      movel([0.367168, -1.380933, -2.569217, -0.762240, 1.570796, 1.937965],accel_mss,speed_ms,0,blend_radius_m)
      movel([0.367388, -1.380879, -2.569255, -0.762256, 1.570796, 1.938184],accel_mss,speed_ms,0,blend_radius_m)
      movel([0.367623, -1.380831, -2.569289, -0.762270, 1.570796, 1.938419],accel_mss,speed_ms,0,blend_radius_m)
      movel([0.367853, -1.380796, -2.569313, -0.762280, 1.570796, 1.938649],accel_mss,speed_ms,0,blend_radius_m)
      movel([0.368080, -1.380773, -2.569329, -0.762287, 1.570796, 1.938877],accel_mss,speed_ms,0,blend_radius_m)
      movel([0.368708, -1.380733, -2.569357, -0.762298, 1.570796, 1.939505],accel_mss,speed_ms,0,blend_radius_m)
      movel([0.369332, -1.380703, -2.569379, -0.762307, 1.570796, 1.940129],accel_mss,speed_ms,0,blend_radius_m)
      movel([0.369955, -1.380682, -2.569394, -0.762313, 1.570796, 1.940751],accel_mss,speed_ms,0,blend_radius_m)
      movel([0.370572, -1.380670, -2.569402, -0.762317, 1.570796, 1.941368],accel_mss,speed_ms,0,blend_radius_m)
      movel([0.370788, -1.380675, -2.569399, -0.762315, 1.570796, 1.941585],accel_mss,speed_ms,0,blend_radius_m)
      movel([0.370998, -1.380691, -2.569387, -0.762311, 1.570796, 1.941795],accel_mss,speed_ms,0,blend_radius_m)
      movel([0.371200, -1.380721, -2.569366, -0.762302, 1.570796, 1.941996],accel_mss,speed_ms,0,blend_radius_m)
      movel([0.371383, -1.380759, -2.569339, -0.762291, 1.570796, 1.942179],accel_mss,speed_ms,0,blend_radius_m)
      movel([0.371557, -1.380812, -2.569302, -0.762275, 1.570796, 1.942353],accel_mss,speed_ms,0,blend_radius_m)
      movel([0.371719, -1.380877, -2.569256, -0.762256, 1.570796, 1.942516],accel_mss,speed_ms,0,blend_radius_m)
      movel([0.372096, -1.381057, -2.569129, -0.762203, 1.570796, 1.942892],accel_mss,speed_ms,0,blend_radius_m)
      movel([0.372463, -1.381249, -2.568993, -0.762147, 1.570796, 1.943259],accel_mss,speed_ms,0,blend_radius_m)
      movel([0.372728, -1.381406, -2.568882, -0.762101, 1.570796, 1.943524],accel_mss,speed_ms,0,blend_radius_m)
      movel([0.372979, -1.381575, -2.568762, -0.762052, 1.570796, 1.943776],accel_mss,speed_ms,0,blend_radius_m)
      movel([0.373219, -1.381756, -2.568634, -0.761999, 1.570796, 1.944015],accel_mss,speed_ms,0,blend_radius_m)
      movel([0.373443, -1.381953, -2.568494, -0.761941, 1.570796, 1.944239],accel_mss,speed_ms,0,blend_radius_m)
      movel([0.373656, -1.382160, -2.568348, -0.761881, 1.570796, 1.944452],accel_mss,speed_ms,0,blend_radius_m)
      movel([0.373848, -1.382378, -2.568193, -0.761818, 1.570796, 1.944644],accel_mss,speed_ms,0,blend_radius_m)
      movel([0.374028, -1.382608, -2.568030, -0.761751, 1.570796, 1.944825],accel_mss,speed_ms,0,blend_radius_m)
      movel([0.374190, -1.382850, -2.567859, -0.761681, 1.570796, 1.944986],accel_mss,speed_ms,0,blend_radius_m)
      movel([0.374338, -1.383103, -2.567679, -0.761607, 1.570796, 1.945134],accel_mss,speed_ms,0,blend_radius_m)
      movel([0.374468, -1.383366, -2.567492, -0.761531, 1.570796, 1.945264],accel_mss,speed_ms,0,blend_radius_m)
      movel([0.374585, -1.383643, -2.567295, -0.761451, 1.570796, 1.945381],accel_mss,speed_ms,0,blend_radius_m)
      movel([0.374684, -1.383931, -2.567090, -0.761368, 1.570796, 1.945480],accel_mss,speed_ms,0,blend_radius_m)
      movel([0.374766, -1.384226, -2.566880, -0.761282, 1.570796, 1.945562],accel_mss,speed_ms,0,blend_radius_m)
      movel([0.374834, -1.384529, -2.566665, -0.761195, 1.570796, 1.945630],accel_mss,speed_ms,0,blend_radius_m)
      movel([0.374881, -1.384841, -2.566442, -0.761105, 1.570796, 1.945678],accel_mss,speed_ms,0,blend_radius_m)
      movel([0.374915, -1.385171, -2.566207, -0.761011, 1.570796, 1.945711],accel_mss,speed_ms,0,blend_radius_m)
      movel([0.374934, -1.385509, -2.565967, -0.760914, 1.570796, 1.945730],accel_mss,speed_ms,0,blend_radius_m)
      movel([0.374935, -1.385851, -2.565722, -0.760816, 1.570796, 1.945731],accel_mss,speed_ms,0,blend_radius_m)
      movel([0.374922, -1.386197, -2.565475, -0.760717, 1.570796, 1.945718],accel_mss,speed_ms,0,blend_radius_m)
      movel([0.374892, -1.386549, -2.565223, -0.760617, 1.570796, 1.945688],accel_mss,speed_ms,0,blend_radius_m)
      movel([0.374857, -1.386821, -2.565029, -0.760539, 1.570796, 1.945653],accel_mss,speed_ms,0,blend_radius_m)
      movel([0.374809, -1.387098, -2.564831, -0.760461, 1.570796, 1.945605],accel_mss,speed_ms,0,blend_radius_m)
      movel([0.374747, -1.387375, -2.564633, -0.760382, 1.570796, 1.945543],accel_mss,speed_ms,0,blend_radius_m)
      movel([0.374671, -1.387656, -2.564431, -0.760302, 1.570796, 1.945468],accel_mss,speed_ms,0,blend_radius_m)
      movel([0.374535, -1.388106, -2.564108, -0.760175, 1.570796, 1.945331],accel_mss,speed_ms,0,blend_radius_m)
      movel([0.374382, -1.388556, -2.563786, -0.760048, 1.570796, 1.945178],accel_mss,speed_ms,0,blend_radius_m)
      movel([0.374215, -1.389008, -2.563461, -0.759920, 1.570796, 1.945011],accel_mss,speed_ms,0,blend_radius_m)
      movel([0.374032, -1.389458, -2.563137, -0.759794, 1.570796, 1.944829],accel_mss,speed_ms,0,blend_radius_m)
      movel([0.373834, -1.389909, -2.562813, -0.759667, 1.570796, 1.944630],accel_mss,speed_ms,0,blend_radius_m)
      movel([0.373623, -1.390357, -2.562490, -0.759542, 1.570796, 1.944419],accel_mss,speed_ms,0,blend_radius_m)
      movel([0.373481, -1.390635, -2.562289, -0.759464, 1.570796, 1.944277],accel_mss,speed_ms,0,blend_radius_m)
      movel([0.373327, -1.390909, -2.562092, -0.759388, 1.570796, 1.944123],accel_mss,speed_ms,0,blend_radius_m)
      movel([0.373162, -1.391181, -2.561896, -0.759312, 1.570796, 1.943958],accel_mss,speed_ms,0,blend_radius_m)
      movel([0.372986, -1.391454, -2.561699, -0.759236, 1.570796, 1.943782],accel_mss,speed_ms,0,blend_radius_m)
      movel([0.372747, -1.391796, -2.561451, -0.759141, 1.570796, 1.943544],accel_mss,speed_ms,0,blend_radius_m)
      movel([0.372498, -1.392137, -2.561205, -0.759047, 1.570796, 1.943295],accel_mss,speed_ms,0,blend_radius_m)
      movel([0.372235, -1.392473, -2.560962, -0.758954, 1.570796, 1.943032],accel_mss,speed_ms,0,blend_radius_m)
      movel([0.371963, -1.392805, -2.560722, -0.758862, 1.570796, 1.942759],accel_mss,speed_ms,0,blend_radius_m)
      movel([0.371681, -1.393131, -2.560486, -0.758772, 1.570796, 1.942478],accel_mss,speed_ms,0,blend_radius_m)
      movel([0.371388, -1.393453, -2.560253, -0.758684, 1.570796, 1.942184],accel_mss,speed_ms,0,blend_radius_m)
      movel([0.371084, -1.393768, -2.560024, -0.758597, 1.570796, 1.941880],accel_mss,speed_ms,0,blend_radius_m)
      movel([0.370782, -1.394067, -2.559806, -0.758515, 1.570796, 1.941578],accel_mss,speed_ms,0,blend_radius_m)
      movel([0.370466, -1.394361, -2.559593, -0.758435, 1.570796, 1.941263],accel_mss,speed_ms,0,blend_radius_m)
      movel([0.370145, -1.394648, -2.559385, -0.758356, 1.570796, 1.940941],accel_mss,speed_ms,0,blend_radius_m)
      movel([0.369814, -1.394924, -2.559184, -0.758281, 1.570796, 1.940610],accel_mss,speed_ms,0,blend_radius_m)
      movel([0.369476, -1.395194, -2.558987, -0.758207, 1.570796, 1.940273],accel_mss,speed_ms,0,blend_radius_m)
      movel([0.369130, -1.395453, -2.558799, -0.758137, 1.570796, 1.939926],accel_mss,speed_ms,0,blend_radius_m)
      movel([0.368780, -1.395704, -2.558616, -0.758069, 1.570796, 1.939577],accel_mss,speed_ms,0,blend_radius_m)
      movel([0.368427, -1.395942, -2.558443, -0.758004, 1.570796, 1.939223],accel_mss,speed_ms,0,blend_radius_m)
      movel([0.368069, -1.396168, -2.558278, -0.757943, 1.570796, 1.938865],accel_mss,speed_ms,0,blend_radius_m)
      movel([0.367709, -1.396384, -2.558121, -0.757884, 1.570796, 1.938505],accel_mss,speed_ms,0,blend_radius_m)
      movel([0.367343, -1.396587, -2.557972, -0.757829, 1.570796, 1.938139],accel_mss,speed_ms,0,blend_radius_m)
      movel([0.366973, -1.396782, -2.557831, -0.757777, 1.570796, 1.937769],accel_mss,speed_ms,0,blend_radius_m)
      movel([0.366600, -1.396963, -2.557698, -0.757728, 1.570796, 1.937396],accel_mss,speed_ms,0,blend_radius_m)
      movel([0.366227, -1.397132, -2.557575, -0.757682, 1.570796, 1.937023],accel_mss,speed_ms,0,blend_radius_m)
      movel([0.365850, -1.397290, -2.557460, -0.757640, 1.570796, 1.936646],accel_mss,speed_ms,0,blend_radius_m)
      movel([0.365473, -1.397434, -2.557354, -0.757601, 1.570796, 1.936270],accel_mss,speed_ms,0,blend_radius_m)
      movel([0.365097, -1.397568, -2.557256, -0.757565, 1.570796, 1.935893],accel_mss,speed_ms,0,blend_radius_m)
      movel([0.364719, -1.397687, -2.557169, -0.757533, 1.570796, 1.935516],accel_mss,speed_ms,0,blend_radius_m)
      movel([0.364343, -1.397793, -2.557092, -0.757504, 1.570796, 1.935139],accel_mss,speed_ms,0,blend_radius_m)
      movel([0.363969, -1.397886, -2.557024, -0.757479, 1.570796, 1.934766],accel_mss,speed_ms,0,blend_radius_m)
      movel([0.363599, -1.397965, -2.556966, -0.757458, 1.570796, 1.934395],accel_mss,speed_ms,0,blend_radius_m)
      movel([0.363252, -1.398025, -2.556922, -0.757442, 1.570796, 1.934048],accel_mss,speed_ms,0,blend_radius_m)
      movel([0.362911, -1.398069, -2.556890, -0.757430, 1.570796, 1.933708],accel_mss,speed_ms,0,blend_radius_m)
      movel([0.362576, -1.398099, -2.556868, -0.757422, 1.570796, 1.933372],accel_mss,speed_ms,0,blend_radius_m)
      movel([0.362245, -1.398113, -2.556858, -0.757418, 1.570796, 1.933042],accel_mss,speed_ms,0,blend_radius_m)
      movel([0.361921, -1.398111, -2.556859, -0.757419, 1.570796, 1.932717],accel_mss,speed_ms,0,blend_radius_m)
      movel([0.361603, -1.398095, -2.556871, -0.757423, 1.570796, 1.932400],accel_mss,speed_ms,0,blend_radius_m)
      movel([0.361295, -1.398062, -2.556895, -0.757432, 1.570796, 1.932092],accel_mss,speed_ms,0,blend_radius_m)
      movel([0.360993, -1.398014, -2.556930, -0.757445, 1.570796, 1.931790],accel_mss,speed_ms,0,blend_radius_m)
      movel([0.360704, -1.397950, -2.556977, -0.757462, 1.570796, 1.931501],accel_mss,speed_ms,0,blend_radius_m)
      movel([0.360408, -1.397869, -2.557036, -0.757484, 1.570796, 1.931204],accel_mss,speed_ms,0,blend_radius_m)
      movel([0.360124, -1.397775, -2.557105, -0.757509, 1.570796, 1.930920],accel_mss,speed_ms,0,blend_radius_m)
      movel([0.359848, -1.397665, -2.557185, -0.757539, 1.570796, 1.930645],accel_mss,speed_ms,0,blend_radius_m)
      movel([0.359584, -1.397544, -2.557274, -0.757571, 1.570796, 1.930380],accel_mss,speed_ms,0,blend_radius_m)
      movel([0.359331, -1.397409, -2.557372, -0.757607, 1.570796, 1.930127],accel_mss,speed_ms,0,blend_radius_m)
      movel([0.359090, -1.397261, -2.557481, -0.757647, 1.570796, 1.929886],accel_mss,speed_ms,0,blend_radius_m)
      movel([0.358861, -1.397102, -2.557597, -0.757690, 1.570796, 1.929657],accel_mss,speed_ms,0,blend_radius_m)
      movel([0.358643, -1.396929, -2.557723, -0.757737, 1.570796, 1.929439],accel_mss,speed_ms,0,blend_radius_m)
      movel([0.358439, -1.396744, -2.557858, -0.757787, 1.570796, 1.929235],accel_mss,speed_ms,0,blend_radius_m)
      movel([0.358240, -1.396540, -2.558007, -0.757842, 1.570796, 1.929036],accel_mss,speed_ms,0,blend_radius_m)
      movel([0.358054, -1.396325, -2.558164, -0.757900, 1.570796, 1.928851],accel_mss,speed_ms,0,blend_radius_m)
      movel([0.357880, -1.396097, -2.558330, -0.757962, 1.570796, 1.928676],accel_mss,speed_ms,0,blend_radius_m)
      movel([0.357724, -1.395859, -2.558504, -0.758027, 1.570796, 1.928520],accel_mss,speed_ms,0,blend_radius_m)
      movel([0.357580, -1.395611, -2.558684, -0.758094, 1.570796, 1.928376],accel_mss,speed_ms,0,blend_radius_m)
      movel([0.357451, -1.395353, -2.558872, -0.758164, 1.570796, 1.928248],accel_mss,speed_ms,0,blend_radius_m)
      movel([0.357335, -1.395086, -2.559066, -0.758237, 1.570796, 1.928131],accel_mss,speed_ms,0,blend_radius_m)
      movel([0.357235, -1.394812, -2.559265, -0.758311, 1.570796, 1.928032],accel_mss,speed_ms,0,blend_radius_m)
      movel([0.357151, -1.394526, -2.559473, -0.758390, 1.570796, 1.927948],accel_mss,speed_ms,0,blend_radius_m)
      movel([0.357072, -1.394192, -2.559716, -0.758481, 1.570796, 1.927869],accel_mss,speed_ms,0,blend_radius_m)
      movel([0.357015, -1.393848, -2.559966, -0.758575, 1.570796, 1.927812],accel_mss,speed_ms,0,blend_radius_m)
      movel([0.356975, -1.393496, -2.560221, -0.758672, 1.570796, 1.927771],accel_mss,speed_ms,0,blend_radius_m)
      movel([0.356953, -1.393135, -2.560483, -0.758771, 1.570796, 1.927750],accel_mss,speed_ms,0,blend_radius_m)
      movel([0.356951, -1.392766, -2.560750, -0.758873, 1.570796, 1.927748],accel_mss,speed_ms,0,blend_radius_m)
      movel([0.356969, -1.392391, -2.561021, -0.758976, 1.570796, 1.927766],accel_mss,speed_ms,0,blend_radius_m)
      movel([0.357005, -1.392011, -2.561296, -0.759082, 1.570796, 1.927802],accel_mss,speed_ms,0,blend_radius_m)
      movel([0.357062, -1.391624, -2.561576, -0.759189, 1.570796, 1.927859],accel_mss,speed_ms,0,blend_radius_m)
      movel([0.357124, -1.391284, -2.561822, -0.759284, 1.570796, 1.927920],accel_mss,speed_ms,0,blend_radius_m)
      movel([0.357196, -1.390939, -2.562071, -0.759380, 1.570796, 1.927992],accel_mss,speed_ms,0,blend_radius_m)
      movel([0.357278, -1.390593, -2.562320, -0.759476, 1.570796, 1.928074],accel_mss,speed_ms,0,blend_radius_m)
      speed_ms = 0.003
      movel([0.357278, -1.393848, -2.563790, -0.754751, 1.570796, 1.928074],accel_mss,speed_ms,0,blend_radius_m)
      speed_ms = 0.007
      movel([0.357356, -1.393564, -2.563996, -0.754829, 1.570796, 1.928153],accel_mss,speed_ms,0,blend_radius_m)
      movel([0.357448, -1.393275, -2.564205, -0.754909, 1.570796, 1.928245],accel_mss,speed_ms,0,blend_radius_m)
      movel([0.357553, -1.392988, -2.564413, -0.754988, 1.570796, 1.928350],accel_mss,speed_ms,0,blend_radius_m)
      movel([0.357672, -1.392700, -2.564621, -0.755068, 1.570796, 1.928469],accel_mss,speed_ms,0,blend_radius_m)
      movel([0.357806, -1.392409, -2.564831, -0.755149, 1.570796, 1.928603],accel_mss,speed_ms,0,blend_radius_m)
      movel([0.357953, -1.392121, -2.565039, -0.755229, 1.570796, 1.928749],accel_mss,speed_ms,0,blend_radius_m)
      movel([0.358142, -1.391770, -2.565292, -0.755327, 1.570796, 1.928938],accel_mss,speed_ms,0,blend_radius_m)
      movel([0.358341, -1.391418, -2.565546, -0.755425, 1.570796, 1.929137],accel_mss,speed_ms,0,blend_radius_m)
      movel([0.358546, -1.391068, -2.565798, -0.755522, 1.570796, 1.929342],accel_mss,speed_ms,0,blend_radius_m)
      movel([0.358793, -1.390674, -2.566082, -0.755633, 1.570796, 1.929589],accel_mss,speed_ms,0,blend_radius_m)
      movel([0.359056, -1.390281, -2.566365, -0.755743, 1.570796, 1.929853],accel_mss,speed_ms,0,blend_radius_m)
      movel([0.359336, -1.389894, -2.566643, -0.755852, 1.570796, 1.930132],accel_mss,speed_ms,0,blend_radius_m)
      movel([0.359627, -1.389510, -2.566919, -0.755960, 1.570796, 1.930424],accel_mss,speed_ms,0,blend_radius_m)
      movel([0.359936, -1.389130, -2.567192, -0.756067, 1.570796, 1.930733],accel_mss,speed_ms,0,blend_radius_m)
      movel([0.360247, -1.388769, -2.567451, -0.756169, 1.570796, 1.931043],accel_mss,speed_ms,0,blend_radius_m)
      movel([0.360574, -1.388414, -2.567705, -0.756269, 1.570796, 1.931370],accel_mss,speed_ms,0,blend_radius_m)
      movel([0.360915, -1.388065, -2.567955, -0.756368, 1.570796, 1.931711],accel_mss,speed_ms,0,blend_radius_m)
      movel([0.361265, -1.387726, -2.568198, -0.756465, 1.570796, 1.932062],accel_mss,speed_ms,0,blend_radius_m)
      movel([0.361629, -1.387396, -2.568435, -0.756559, 1.570796, 1.932425],accel_mss,speed_ms,0,blend_radius_m)
      movel([0.361998, -1.387082, -2.568659, -0.756648, 1.570796, 1.932794],accel_mss,speed_ms,0,blend_radius_m)
      movel([0.362374, -1.386777, -2.568876, -0.756735, 1.570796, 1.933171],accel_mss,speed_ms,0,blend_radius_m)
      movel([0.362763, -1.386485, -2.569085, -0.756819, 1.570796, 1.933559],accel_mss,speed_ms,0,blend_radius_m)
      movel([0.363157, -1.386205, -2.569285, -0.756899, 1.570796, 1.933954],accel_mss,speed_ms,0,blend_radius_m)
      movel([0.363562, -1.385937, -2.569476, -0.756976, 1.570796, 1.934358],accel_mss,speed_ms,0,blend_radius_m)
      movel([0.363972, -1.385683, -2.569657, -0.757049, 1.570796, 1.934768],accel_mss,speed_ms,0,blend_radius_m)
      movel([0.364386, -1.385443, -2.569828, -0.757118, 1.570796, 1.935183],accel_mss,speed_ms,0,blend_radius_m)
      movel([0.364807, -1.385215, -2.569990, -0.757183, 1.570796, 1.935604],accel_mss,speed_ms,0,blend_radius_m)
      movel([0.365231, -1.385005, -2.570140, -0.757244, 1.570796, 1.936027],accel_mss,speed_ms,0,blend_radius_m)
      movel([0.365658, -1.384809, -2.570280, -0.757301, 1.570796, 1.936454],accel_mss,speed_ms,0,blend_radius_m)
      movel([0.366192, -1.384581, -2.570442, -0.757366, 1.570796, 1.936988],accel_mss,speed_ms,0,blend_radius_m)
      movel([0.366727, -1.384364, -2.570596, -0.757429, 1.570796, 1.937523],accel_mss,speed_ms,0,blend_radius_m)
      movel([0.366947, -1.384283, -2.570653, -0.757452, 1.570796, 1.937744],accel_mss,speed_ms,0,blend_radius_m)
      movel([0.367168, -1.384214, -2.570703, -0.757473, 1.570796, 1.937965],accel_mss,speed_ms,0,blend_radius_m)
      movel([0.367388, -1.384160, -2.570741, -0.757488, 1.570796, 1.938184],accel_mss,speed_ms,0,blend_radius_m)
      movel([0.367623, -1.384112, -2.570775, -0.757502, 1.570796, 1.938419],accel_mss,speed_ms,0,blend_radius_m)
      movel([0.367853, -1.384078, -2.570799, -0.757512, 1.570796, 1.938649],accel_mss,speed_ms,0,blend_radius_m)
      movel([0.368080, -1.384055, -2.570816, -0.757519, 1.570796, 1.938877],accel_mss,speed_ms,0,blend_radius_m)
      movel([0.368708, -1.384015, -2.570844, -0.757530, 1.570796, 1.939505],accel_mss,speed_ms,0,blend_radius_m)
      movel([0.369332, -1.383985, -2.570865, -0.757539, 1.570796, 1.940129],accel_mss,speed_ms,0,blend_radius_m)
      movel([0.369955, -1.383964, -2.570880, -0.757545, 1.570796, 1.940751],accel_mss,speed_ms,0,blend_radius_m)
      movel([0.370572, -1.383952, -2.570888, -0.757548, 1.570796, 1.941368],accel_mss,speed_ms,0,blend_radius_m)
      movel([0.370788, -1.383957, -2.570885, -0.757547, 1.570796, 1.941585],accel_mss,speed_ms,0,blend_radius_m)
      movel([0.370998, -1.383973, -2.570874, -0.757542, 1.570796, 1.941795],accel_mss,speed_ms,0,blend_radius_m)
      movel([0.371200, -1.384003, -2.570852, -0.757534, 1.570796, 1.941996],accel_mss,speed_ms,0,blend_radius_m)
      movel([0.371383, -1.384040, -2.570826, -0.757523, 1.570796, 1.942179],accel_mss,speed_ms,0,blend_radius_m)
      movel([0.371557, -1.384094, -2.570788, -0.757507, 1.570796, 1.942353],accel_mss,speed_ms,0,blend_radius_m)
      movel([0.371719, -1.384159, -2.570742, -0.757489, 1.570796, 1.942516],accel_mss,speed_ms,0,blend_radius_m)
      movel([0.372096, -1.384338, -2.570614, -0.757437, 1.570796, 1.942892],accel_mss,speed_ms,0,blend_radius_m)
      movel([0.372463, -1.384529, -2.570479, -0.757381, 1.570796, 1.943259],accel_mss,speed_ms,0,blend_radius_m)
      movel([0.372728, -1.384686, -2.570367, -0.757336, 1.570796, 1.943524],accel_mss,speed_ms,0,blend_radius_m)
      movel([0.372979, -1.384855, -2.570247, -0.757287, 1.570796, 1.943776],accel_mss,speed_ms,0,blend_radius_m)
      movel([0.373219, -1.385035, -2.570119, -0.757235, 1.570796, 1.944015],accel_mss,speed_ms,0,blend_radius_m)
      movel([0.373443, -1.385231, -2.569979, -0.757179, 1.570796, 1.944239],accel_mss,speed_ms,0,blend_radius_m)
      movel([0.373656, -1.385437, -2.569832, -0.757119, 1.570796, 1.944452],accel_mss,speed_ms,0,blend_radius_m)
      movel([0.373848, -1.385655, -2.569677, -0.757057, 1.570796, 1.944644],accel_mss,speed_ms,0,blend_radius_m)
      movel([0.374028, -1.385884, -2.569514, -0.756991, 1.570796, 1.944825],accel_mss,speed_ms,0,blend_radius_m)
      movel([0.374190, -1.386126, -2.569342, -0.756922, 1.570796, 1.944986],accel_mss,speed_ms,0,blend_radius_m)
      movel([0.374338, -1.386378, -2.569161, -0.756849, 1.570796, 1.945134],accel_mss,speed_ms,0,blend_radius_m)
      movel([0.374468, -1.386640, -2.568974, -0.756774, 1.570796, 1.945264],accel_mss,speed_ms,0,blend_radius_m)
      movel([0.374585, -1.386916, -2.568777, -0.756696, 1.570796, 1.945381],accel_mss,speed_ms,0,blend_radius_m)
      movel([0.374684, -1.387204, -2.568572, -0.756613, 1.570796, 1.945480],accel_mss,speed_ms,0,blend_radius_m)
      movel([0.374766, -1.387499, -2.568361, -0.756529, 1.570796, 1.945562],accel_mss,speed_ms,0,blend_radius_m)
      movel([0.374834, -1.387800, -2.568145, -0.756444, 1.570796, 1.945630],accel_mss,speed_ms,0,blend_radius_m)
      movel([0.374881, -1.388112, -2.567922, -0.756355, 1.570796, 1.945678],accel_mss,speed_ms,0,blend_radius_m)
      movel([0.374915, -1.388441, -2.567686, -0.756262, 1.570796, 1.945711],accel_mss,speed_ms,0,blend_radius_m)
      movel([0.374934, -1.388777, -2.567445, -0.756167, 1.570796, 1.945730],accel_mss,speed_ms,0,blend_radius_m)
      movel([0.374935, -1.389118, -2.567200, -0.756070, 1.570796, 1.945731],accel_mss,speed_ms,0,blend_radius_m)
      movel([0.374922, -1.389464, -2.566952, -0.755973, 1.570796, 1.945718],accel_mss,speed_ms,0,blend_radius_m)
      movel([0.374892, -1.389815, -2.566700, -0.755874, 1.570796, 1.945688],accel_mss,speed_ms,0,blend_radius_m)
      movel([0.374857, -1.390086, -2.566505, -0.755798, 1.570796, 1.945653],accel_mss,speed_ms,0,blend_radius_m)
      movel([0.374809, -1.390362, -2.566307, -0.755720, 1.570796, 1.945605],accel_mss,speed_ms,0,blend_radius_m)
      movel([0.374747, -1.390638, -2.566108, -0.755643, 1.570796, 1.945543],accel_mss,speed_ms,0,blend_radius_m)
      movel([0.374671, -1.390919, -2.565906, -0.755564, 1.570796, 1.945468],accel_mss,speed_ms,0,blend_radius_m)
      movel([0.374535, -1.391367, -2.565583, -0.755439, 1.570796, 1.945331],accel_mss,speed_ms,0,blend_radius_m)
      movel([0.374382, -1.391816, -2.565259, -0.755314, 1.570796, 1.945178],accel_mss,speed_ms,0,blend_radius_m)
      movel([0.374215, -1.392267, -2.564934, -0.755188, 1.570796, 1.945011],accel_mss,speed_ms,0,blend_radius_m)
      movel([0.374032, -1.392716, -2.564609, -0.755064, 1.570796, 1.944829],accel_mss,speed_ms,0,blend_radius_m)
      movel([0.373834, -1.393165, -2.564284, -0.754939, 1.570796, 1.944630],accel_mss,speed_ms,0,blend_radius_m)
      movel([0.373623, -1.393612, -2.563961, -0.754816, 1.570796, 1.944419],accel_mss,speed_ms,0,blend_radius_m)
      movel([0.373481, -1.393890, -2.563760, -0.754739, 1.570796, 1.944277],accel_mss,speed_ms,0,blend_radius_m)
      movel([0.373327, -1.394163, -2.563562, -0.754664, 1.570796, 1.944123],accel_mss,speed_ms,0,blend_radius_m)
      movel([0.373162, -1.394434, -2.563365, -0.754590, 1.570796, 1.943958],accel_mss,speed_ms,0,blend_radius_m)
      movel([0.372986, -1.394706, -2.563168, -0.754515, 1.570796, 1.943782],accel_mss,speed_ms,0,blend_radius_m)
      movel([0.372747, -1.395048, -2.562920, -0.754422, 1.570796, 1.943544],accel_mss,speed_ms,0,blend_radius_m)
      movel([0.372498, -1.395387, -2.562673, -0.754329, 1.570796, 1.943295],accel_mss,speed_ms,0,blend_radius_m)
      movel([0.372235, -1.395723, -2.562429, -0.754237, 1.570796, 1.943032],accel_mss,speed_ms,0,blend_radius_m)
      movel([0.371963, -1.396054, -2.562188, -0.754147, 1.570796, 1.942759],accel_mss,speed_ms,0,blend_radius_m)
      movel([0.371681, -1.396379, -2.561952, -0.754058, 1.570796, 1.942478],accel_mss,speed_ms,0,blend_radius_m)
      movel([0.371388, -1.396699, -2.561718, -0.753971, 1.570796, 1.942184],accel_mss,speed_ms,0,blend_radius_m)
      movel([0.371084, -1.397014, -2.561489, -0.753886, 1.570796, 1.941880],accel_mss,speed_ms,0,blend_radius_m)
      movel([0.370782, -1.397313, -2.561271, -0.753805, 1.570796, 1.941578],accel_mss,speed_ms,0,blend_radius_m)
      movel([0.370466, -1.397605, -2.561058, -0.753726, 1.570796, 1.941263],accel_mss,speed_ms,0,blend_radius_m)
      movel([0.370145, -1.397892, -2.560848, -0.753649, 1.570796, 1.940941],accel_mss,speed_ms,0,blend_radius_m)
      movel([0.369814, -1.398167, -2.560647, -0.753575, 1.570796, 1.940610],accel_mss,speed_ms,0,blend_radius_m)
      movel([0.369476, -1.398436, -2.560450, -0.753502, 1.570796, 1.940273],accel_mss,speed_ms,0,blend_radius_m)
      movel([0.369130, -1.398695, -2.560261, -0.753433, 1.570796, 1.939926],accel_mss,speed_ms,0,blend_radius_m)
      movel([0.368780, -1.398945, -2.560078, -0.753366, 1.570796, 1.939577],accel_mss,speed_ms,0,blend_radius_m)
      movel([0.368427, -1.399182, -2.559905, -0.753302, 1.570796, 1.939223],accel_mss,speed_ms,0,blend_radius_m)
      movel([0.368069, -1.399408, -2.559739, -0.753242, 1.570796, 1.938865],accel_mss,speed_ms,0,blend_radius_m)
      movel([0.367709, -1.399623, -2.559582, -0.753184, 1.570796, 1.938505],accel_mss,speed_ms,0,blend_radius_m)
      movel([0.367343, -1.399826, -2.559433, -0.753130, 1.570796, 1.938139],accel_mss,speed_ms,0,blend_radius_m)
      movel([0.366973, -1.400019, -2.559291, -0.753079, 1.570796, 1.937769],accel_mss,speed_ms,0,blend_radius_m)
      movel([0.366600, -1.400201, -2.559158, -0.753030, 1.570796, 1.937396],accel_mss,speed_ms,0,blend_radius_m)
      movel([0.366227, -1.400369, -2.559035, -0.752986, 1.570796, 1.937023],accel_mss,speed_ms,0,blend_radius_m)
      movel([0.365850, -1.400526, -2.558919, -0.752944, 1.570796, 1.936646],accel_mss,speed_ms,0,blend_radius_m)
      movel([0.365473, -1.400670, -2.558813, -0.752906, 1.570796, 1.936270],accel_mss,speed_ms,0,blend_radius_m)
      movel([0.365097, -1.400804, -2.558715, -0.752870, 1.570796, 1.935893],accel_mss,speed_ms,0,blend_radius_m)
      movel([0.364719, -1.400922, -2.558628, -0.752839, 1.570796, 1.935516],accel_mss,speed_ms,0,blend_radius_m)
      movel([0.364343, -1.401028, -2.558550, -0.752811, 1.570796, 1.935139],accel_mss,speed_ms,0,blend_radius_m)
      movel([0.363969, -1.401120, -2.558482, -0.752786, 1.570796, 1.934766],accel_mss,speed_ms,0,blend_radius_m)
      movel([0.363599, -1.401200, -2.558424, -0.752765, 1.570796, 1.934395],accel_mss,speed_ms,0,blend_radius_m)
      movel([0.363252, -1.401259, -2.558381, -0.752749, 1.570796, 1.934048],accel_mss,speed_ms,0,blend_radius_m)
      movel([0.362911, -1.401303, -2.558348, -0.752738, 1.570796, 1.933708],accel_mss,speed_ms,0,blend_radius_m)
      movel([0.362576, -1.401333, -2.558326, -0.752730, 1.570796, 1.933372],accel_mss,speed_ms,0,blend_radius_m)
      movel([0.362245, -1.401347, -2.558316, -0.752726, 1.570796, 1.933042],accel_mss,speed_ms,0,blend_radius_m)
      movel([0.361921, -1.401345, -2.558318, -0.752727, 1.570796, 1.932717],accel_mss,speed_ms,0,blend_radius_m)
      movel([0.361603, -1.401329, -2.558329, -0.752731, 1.570796, 1.932400],accel_mss,speed_ms,0,blend_radius_m)
      movel([0.361295, -1.401297, -2.558353, -0.752740, 1.570796, 1.932092],accel_mss,speed_ms,0,blend_radius_m)
      movel([0.360993, -1.401248, -2.558388, -0.752752, 1.570796, 1.931790],accel_mss,speed_ms,0,blend_radius_m)
      movel([0.360704, -1.401185, -2.558435, -0.752769, 1.570796, 1.931501],accel_mss,speed_ms,0,blend_radius_m)
      movel([0.360408, -1.401104, -2.558495, -0.752791, 1.570796, 1.931204],accel_mss,speed_ms,0,blend_radius_m)
      movel([0.360124, -1.401010, -2.558564, -0.752815, 1.570796, 1.930920],accel_mss,speed_ms,0,blend_radius_m)
      movel([0.359848, -1.400900, -2.558644, -0.752845, 1.570796, 1.930645],accel_mss,speed_ms,0,blend_radius_m)
      movel([0.359584, -1.400779, -2.558733, -0.752877, 1.570796, 1.930380],accel_mss,speed_ms,0,blend_radius_m)
      movel([0.359331, -1.400645, -2.558832, -0.752912, 1.570796, 1.930127],accel_mss,speed_ms,0,blend_radius_m)
      movel([0.359090, -1.400497, -2.558940, -0.752951, 1.570796, 1.929886],accel_mss,speed_ms,0,blend_radius_m)
      movel([0.358861, -1.400338, -2.559057, -0.752994, 1.570796, 1.929657],accel_mss,speed_ms,0,blend_radius_m)
      movel([0.358643, -1.400166, -2.559183, -0.753040, 1.570796, 1.929439],accel_mss,speed_ms,0,blend_radius_m)
      movel([0.358439, -1.399982, -2.559318, -0.753089, 1.570796, 1.929235],accel_mss,speed_ms,0,blend_radius_m)
      movel([0.358240, -1.399778, -2.559468, -0.753143, 1.570796, 1.929036],accel_mss,speed_ms,0,blend_radius_m)
      movel([0.358054, -1.399563, -2.559625, -0.753200, 1.570796, 1.928851],accel_mss,speed_ms,0,blend_radius_m)
      movel([0.357880, -1.399337, -2.559791, -0.753261, 1.570796, 1.928676],accel_mss,speed_ms,0,blend_radius_m)
      movel([0.357724, -1.399099, -2.559966, -0.753325, 1.570796, 1.928520],accel_mss,speed_ms,0,blend_radius_m)
      movel([0.357580, -1.398852, -2.560147, -0.753391, 1.570796, 1.928376],accel_mss,speed_ms,0,blend_radius_m)
      movel([0.357451, -1.398595, -2.560334, -0.753460, 1.570796, 1.928248],accel_mss,speed_ms,0,blend_radius_m)
      movel([0.357335, -1.398329, -2.560529, -0.753531, 1.570796, 1.928131],accel_mss,speed_ms,0,blend_radius_m)
      movel([0.357235, -1.398055, -2.560729, -0.753605, 1.570796, 1.928032],accel_mss,speed_ms,0,blend_radius_m)
      movel([0.357151, -1.397770, -2.560937, -0.753682, 1.570796, 1.927948],accel_mss,speed_ms,0,blend_radius_m)
      movel([0.357072, -1.397437, -2.561180, -0.753772, 1.570796, 1.927869],accel_mss,speed_ms,0,blend_radius_m)
      movel([0.357015, -1.397094, -2.561431, -0.753864, 1.570796, 1.927812],accel_mss,speed_ms,0,blend_radius_m)
      movel([0.356975, -1.396743, -2.561686, -0.753959, 1.570796, 1.927771],accel_mss,speed_ms,0,blend_radius_m)
      movel([0.356953, -1.396383, -2.561949, -0.754057, 1.570796, 1.927750],accel_mss,speed_ms,0,blend_radius_m)
      movel([0.356951, -1.396015, -2.562217, -0.754157, 1.570796, 1.927748],accel_mss,speed_ms,0,blend_radius_m)
      movel([0.356969, -1.395641, -2.562488, -0.754259, 1.570796, 1.927766],accel_mss,speed_ms,0,blend_radius_m)
      movel([0.357005, -1.395262, -2.562764, -0.754363, 1.570796, 1.927802],accel_mss,speed_ms,0,blend_radius_m)
      movel([0.357062, -1.394876, -2.563045, -0.754469, 1.570796, 1.927859],accel_mss,speed_ms,0,blend_radius_m)
      movel([0.357124, -1.394536, -2.563291, -0.754562, 1.570796, 1.927920],accel_mss,speed_ms,0,blend_radius_m)
      movel([0.357196, -1.394192, -2.563540, -0.754656, 1.570796, 1.927992],accel_mss,speed_ms,0,blend_radius_m)
      movel([0.357278, -1.393848, -2.563790, -0.754751, 1.570796, 1.928074],accel_mss,speed_ms,0,blend_radius_m)
      speed_ms = 0.003
      movel([0.357278, -1.380960, -2.557859, -0.773571, 1.570796, 1.928074],accel_mss,speed_ms,0,blend_radius_m)
      speed_ms = 0.01
      movel([0.357278, -1.356224, -2.545602, -0.810563, 1.570796, 1.928074],accel_mss,speed_ms,0,blend_radius_m)
      movel([0.358426, -1.356634, -2.545321, -0.810434, 1.570796, 1.929222],accel_mss,speed_ms,0,blend_radius_m)
      movel([0.358426, -1.381362, -2.557573, -0.773455, 1.570796, 1.929222],accel_mss,speed_ms,0,blend_radius_m)
      speed_ms = 0.003
      movel([0.358426, -1.390992, -2.562032, -0.759365, 1.570796, 1.929222],accel_mss,speed_ms,0,blend_radius_m)
      speed_ms = 0.007
      movel([0.358674, -1.390327, -2.562512, -0.759550, 1.570796, 1.929470],accel_mss,speed_ms,0,blend_radius_m)
      movel([0.358928, -1.389663, -2.562990, -0.759736, 1.570796, 1.929724],accel_mss,speed_ms,0,blend_radius_m)
      movel([0.359196, -1.388987, -2.563476, -0.759926, 1.570796, 1.929992],accel_mss,speed_ms,0,blend_radius_m)
      movel([0.359471, -1.388309, -2.563962, -0.760117, 1.570796, 1.930267],accel_mss,speed_ms,0,blend_radius_m)
      movel([0.359570, -1.388085, -2.564124, -0.760181, 1.570796, 1.930367],accel_mss,speed_ms,0,blend_radius_m)
      movel([0.359681, -1.387859, -2.564285, -0.760244, 1.570796, 1.930477],accel_mss,speed_ms,0,blend_radius_m)
      movel([0.359803, -1.387636, -2.564446, -0.760308, 1.570796, 1.930599],accel_mss,speed_ms,0,blend_radius_m)
      movel([0.359919, -1.387443, -2.564584, -0.760363, 1.570796, 1.930715],accel_mss,speed_ms,0,blend_radius_m)
      movel([0.360048, -1.387254, -2.564719, -0.760416, 1.570796, 1.930844],accel_mss,speed_ms,0,blend_radius_m)
      movel([0.360189, -1.387069, -2.564852, -0.760469, 1.570796, 1.930985],accel_mss,speed_ms,0,blend_radius_m)
      movel([0.360518, -1.386665, -2.565140, -0.760584, 1.570796, 1.931314],accel_mss,speed_ms,0,blend_radius_m)
      movel([0.360858, -1.386269, -2.565423, -0.760696, 1.570796, 1.931654],accel_mss,speed_ms,0,blend_radius_m)
      movel([0.361119, -1.385981, -2.565629, -0.760779, 1.570796, 1.931916],accel_mss,speed_ms,0,blend_radius_m)
      movel([0.361388, -1.385699, -2.565831, -0.760859, 1.570796, 1.932184],accel_mss,speed_ms,0,blend_radius_m)
      movel([0.361665, -1.385423, -2.566028, -0.760938, 1.570796, 1.932462],accel_mss,speed_ms,0,blend_radius_m)
      movel([0.361951, -1.385151, -2.566222, -0.761016, 1.570796, 1.932747],accel_mss,speed_ms,0,blend_radius_m)
      movel([0.362243, -1.384890, -2.566408, -0.761091, 1.570796, 1.933040],accel_mss,speed_ms,0,blend_radius_m)
      movel([0.362544, -1.384632, -2.566591, -0.761165, 1.570796, 1.933340],accel_mss,speed_ms,0,blend_radius_m)
      movel([0.362850, -1.384383, -2.566769, -0.761237, 1.570796, 1.933646],accel_mss,speed_ms,0,blend_radius_m)
      movel([0.363162, -1.384143, -2.566940, -0.761306, 1.570796, 1.933959],accel_mss,speed_ms,0,blend_radius_m)
      movel([0.363474, -1.383916, -2.567101, -0.761372, 1.570796, 1.934270],accel_mss,speed_ms,0,blend_radius_m)
      movel([0.363789, -1.383698, -2.567256, -0.761435, 1.570796, 1.934586],accel_mss,speed_ms,0,blend_radius_m)
      movel([0.364110, -1.383490, -2.567404, -0.761495, 1.570796, 1.934906],accel_mss,speed_ms,0,blend_radius_m)
      movel([0.364437, -1.383289, -2.567547, -0.761553, 1.570796, 1.935233],accel_mss,speed_ms,0,blend_radius_m)
      movel([0.364752, -1.383108, -2.567675, -0.761606, 1.570796, 1.935548],accel_mss,speed_ms,0,blend_radius_m)
      movel([0.365072, -1.382936, -2.567797, -0.761655, 1.570796, 1.935868],accel_mss,speed_ms,0,blend_radius_m)
      movel([0.365394, -1.382778, -2.567910, -0.761702, 1.570796, 1.936190],accel_mss,speed_ms,0,blend_radius_m)
      movel([0.365717, -1.382630, -2.568014, -0.761744, 1.570796, 1.936513],accel_mss,speed_ms,0,blend_radius_m)
      movel([0.366119, -1.382461, -2.568134, -0.761793, 1.570796, 1.936915],accel_mss,speed_ms,0,blend_radius_m)
      movel([0.366520, -1.382306, -2.568244, -0.761839, 1.570796, 1.937316],accel_mss,speed_ms,0,blend_radius_m)
      movel([0.366722, -1.382237, -2.568293, -0.761859, 1.570796, 1.937518],accel_mss,speed_ms,0,blend_radius_m)
      movel([0.366925, -1.382177, -2.568335, -0.761876, 1.570796, 1.937721],accel_mss,speed_ms,0,blend_radius_m)
      movel([0.367125, -1.382131, -2.568368, -0.761890, 1.570796, 1.937921],accel_mss,speed_ms,0,blend_radius_m)
      movel([0.367346, -1.382088, -2.568399, -0.761902, 1.570796, 1.938143],accel_mss,speed_ms,0,blend_radius_m)
      movel([0.367566, -1.382057, -2.568421, -0.761911, 1.570796, 1.938362],accel_mss,speed_ms,0,blend_radius_m)
      movel([0.367783, -1.382036, -2.568435, -0.761917, 1.570796, 1.938579],accel_mss,speed_ms,0,blend_radius_m)
      movel([0.368308, -1.381999, -2.568462, -0.761928, 1.570796, 1.939104],accel_mss,speed_ms,0,blend_radius_m)
      movel([0.368831, -1.381973, -2.568481, -0.761936, 1.570796, 1.939627],accel_mss,speed_ms,0,blend_radius_m)
      movel([0.369362, -1.381955, -2.568493, -0.761941, 1.570796, 1.940158],accel_mss,speed_ms,0,blend_radius_m)
      movel([0.369888, -1.381950, -2.568497, -0.761943, 1.570796, 1.940684],accel_mss,speed_ms,0,blend_radius_m)
      movel([0.370095, -1.381955, -2.568493, -0.761941, 1.570796, 1.940891],accel_mss,speed_ms,0,blend_radius_m)
      movel([0.370296, -1.381969, -2.568483, -0.761937, 1.570796, 1.941092],accel_mss,speed_ms,0,blend_radius_m)
      movel([0.370489, -1.381997, -2.568463, -0.761929, 1.570796, 1.941285],accel_mss,speed_ms,0,blend_radius_m)
      movel([0.370661, -1.382032, -2.568438, -0.761918, 1.570796, 1.941457],accel_mss,speed_ms,0,blend_radius_m)
      movel([0.370825, -1.382082, -2.568403, -0.761904, 1.570796, 1.941621],accel_mss,speed_ms,0,blend_radius_m)
      movel([0.370983, -1.382140, -2.568362, -0.761887, 1.570796, 1.941779],accel_mss,speed_ms,0,blend_radius_m)
      movel([0.371305, -1.382288, -2.568257, -0.761844, 1.570796, 1.942101],accel_mss,speed_ms,0,blend_radius_m)
      movel([0.371615, -1.382448, -2.568144, -0.761797, 1.570796, 1.942412],accel_mss,speed_ms,0,blend_radius_m)
      movel([0.371844, -1.382582, -2.568049, -0.761758, 1.570796, 1.942640],accel_mss,speed_ms,0,blend_radius_m)
      movel([0.372062, -1.382730, -2.567944, -0.761716, 1.570796, 1.942859],accel_mss,speed_ms,0,blend_radius_m)
      movel([0.372266, -1.382891, -2.567829, -0.761669, 1.570796, 1.943062],accel_mss,speed_ms,0,blend_radius_m)
      movel([0.372459, -1.383062, -2.567708, -0.761619, 1.570796, 1.943255],accel_mss,speed_ms,0,blend_radius_m)
      movel([0.372637, -1.383247, -2.567576, -0.761565, 1.570796, 1.943433],accel_mss,speed_ms,0,blend_radius_m)
      movel([0.372801, -1.383444, -2.567437, -0.761508, 1.570796, 1.943597],accel_mss,speed_ms,0,blend_radius_m)
      movel([0.372948, -1.383652, -2.567289, -0.761448, 1.570796, 1.943745],accel_mss,speed_ms,0,blend_radius_m)
      movel([0.373083, -1.383870, -2.567134, -0.761385, 1.570796, 1.943879],accel_mss,speed_ms,0,blend_radius_m)
      movel([0.373225, -1.384138, -2.566943, -0.761308, 1.570796, 1.944021],accel_mss,speed_ms,0,blend_radius_m)
      movel([0.373345, -1.384419, -2.566743, -0.761227, 1.570796, 1.944142],accel_mss,speed_ms,0,blend_radius_m)
      movel([0.373450, -1.384711, -2.566535, -0.761143, 1.570796, 1.944246],accel_mss,speed_ms,0,blend_radius_m)
      movel([0.373533, -1.385015, -2.566319, -0.761056, 1.570796, 1.944329],accel_mss,speed_ms,0,blend_radius_m)
      movel([0.373597, -1.385328, -2.566095, -0.760966, 1.570796, 1.944393],accel_mss,speed_ms,0,blend_radius_m)
      movel([0.373641, -1.385649, -2.565867, -0.760874, 1.570796, 1.944437],accel_mss,speed_ms,0,blend_radius_m)
      movel([0.373668, -1.385978, -2.565631, -0.760779, 1.570796, 1.944464],accel_mss,speed_ms,0,blend_radius_m)
      movel([0.373674, -1.386320, -2.565387, -0.760682, 1.570796, 1.944470],accel_mss,speed_ms,0,blend_radius_m)
      movel([0.373659, -1.386669, -2.565138, -0.760583, 1.570796, 1.944455],accel_mss,speed_ms,0,blend_radius_m)
      movel([0.373627, -1.387024, -2.564883, -0.760481, 1.570796, 1.944423],accel_mss,speed_ms,0,blend_radius_m)
      movel([0.373576, -1.387383, -2.564626, -0.760379, 1.570796, 1.944372],accel_mss,speed_ms,0,blend_radius_m)
      movel([0.373503, -1.387749, -2.564364, -0.760276, 1.570796, 1.944300],accel_mss,speed_ms,0,blend_radius_m)
      movel([0.373412, -1.388115, -2.564102, -0.760172, 1.570796, 1.944209],accel_mss,speed_ms,0,blend_radius_m)
      movel([0.373304, -1.388486, -2.563836, -0.760067, 1.570796, 1.944100],accel_mss,speed_ms,0,blend_radius_m)
      movel([0.373175, -1.388855, -2.563571, -0.759963, 1.570796, 1.943971],accel_mss,speed_ms,0,blend_radius_m)
      movel([0.373030, -1.389224, -2.563305, -0.759859, 1.570796, 1.943827],accel_mss,speed_ms,0,blend_radius_m)
      movel([0.372866, -1.389597, -2.563037, -0.759755, 1.570796, 1.943663],accel_mss,speed_ms,0,blend_radius_m)
      movel([0.372686, -1.389965, -2.562773, -0.759652, 1.570796, 1.943482],accel_mss,speed_ms,0,blend_radius_m)
      movel([0.372487, -1.390333, -2.562507, -0.759549, 1.570796, 1.943283],accel_mss,speed_ms,0,blend_radius_m)
      movel([0.372271, -1.390700, -2.562243, -0.759446, 1.570796, 1.943067],accel_mss,speed_ms,0,blend_radius_m)
      movel([0.372039, -1.391060, -2.561983, -0.759346, 1.570796, 1.942835],accel_mss,speed_ms,0,blend_radius_m)
      movel([0.371814, -1.391385, -2.561748, -0.759255, 1.570796, 1.942611],accel_mss,speed_ms,0,blend_radius_m)
      movel([0.371581, -1.391706, -2.561517, -0.759166, 1.570796, 1.942377],accel_mss,speed_ms,0,blend_radius_m)
      movel([0.371333, -1.392022, -2.561288, -0.759079, 1.570796, 1.942129],accel_mss,speed_ms,0,blend_radius_m)
      movel([0.371076, -1.392332, -2.561064, -0.758993, 1.570796, 1.941872],accel_mss,speed_ms,0,blend_radius_m)
      movel([0.370810, -1.392638, -2.560843, -0.758908, 1.570796, 1.941606],accel_mss,speed_ms,0,blend_radius_m)
      movel([0.370537, -1.392933, -2.560629, -0.758827, 1.570796, 1.941333],accel_mss,speed_ms,0,blend_radius_m)
      movel([0.370253, -1.393219, -2.560422, -0.758748, 1.570796, 1.941050],accel_mss,speed_ms,0,blend_radius_m)
      movel([0.369963, -1.393497, -2.560220, -0.758672, 1.570796, 1.940759],accel_mss,speed_ms,0,blend_radius_m)
      movel([0.369663, -1.393769, -2.560023, -0.758597, 1.570796, 1.940459],accel_mss,speed_ms,0,blend_radius_m)
      movel([0.369355, -1.394032, -2.559832, -0.758525, 1.570796, 1.940152],accel_mss,speed_ms,0,blend_radius_m)
      movel([0.369041, -1.394284, -2.559649, -0.758456, 1.570796, 1.939837],accel_mss,speed_ms,0,blend_radius_m)
      movel([0.368722, -1.394525, -2.559474, -0.758390, 1.570796, 1.939518],accel_mss,speed_ms,0,blend_radius_m)
      movel([0.368395, -1.394758, -2.559305, -0.758326, 1.570796, 1.939192],accel_mss,speed_ms,0,blend_radius_m)
      movel([0.368064, -1.394980, -2.559144, -0.758266, 1.570796, 1.938860],accel_mss,speed_ms,0,blend_radius_m)
      movel([0.367728, -1.395191, -2.558990, -0.758208, 1.570796, 1.938524],accel_mss,speed_ms,0,blend_radius_m)
      movel([0.367387, -1.395391, -2.558844, -0.758154, 1.570796, 1.938184],accel_mss,speed_ms,0,blend_radius_m)
      movel([0.367040, -1.395581, -2.558706, -0.758102, 1.570796, 1.937836],accel_mss,speed_ms,0,blend_radius_m)
      movel([0.366693, -1.395758, -2.558577, -0.758054, 1.570796, 1.937489],accel_mss,speed_ms,0,blend_radius_m)
      movel([0.366341, -1.395924, -2.558456, -0.758009, 1.570796, 1.937138],accel_mss,speed_ms,0,blend_radius_m)
      movel([0.365988, -1.396077, -2.558345, -0.757967, 1.570796, 1.936785],accel_mss,speed_ms,0,blend_radius_m)
      movel([0.365621, -1.396221, -2.558239, -0.757928, 1.570796, 1.936417],accel_mss,speed_ms,0,blend_radius_m)
      movel([0.365251, -1.396353, -2.558143, -0.757892, 1.570796, 1.936047],accel_mss,speed_ms,0,blend_radius_m)
      movel([0.365052, -1.396415, -2.558098, -0.757876, 1.570796, 1.935848],accel_mss,speed_ms,0,blend_radius_m)
      movel([0.364854, -1.396469, -2.558059, -0.757861, 1.570796, 1.935651],accel_mss,speed_ms,0,blend_radius_m)
      movel([0.364658, -1.396514, -2.558026, -0.757849, 1.570796, 1.935454],accel_mss,speed_ms,0,blend_radius_m)
      movel([0.364437, -1.396550, -2.557999, -0.757839, 1.570796, 1.935233],accel_mss,speed_ms,0,blend_radius_m)
      movel([0.364217, -1.396581, -2.557977, -0.757831, 1.570796, 1.935013],accel_mss,speed_ms,0,blend_radius_m)
      movel([0.364000, -1.396602, -2.557961, -0.757825, 1.570796, 1.934796],accel_mss,speed_ms,0,blend_radius_m)
      movel([0.363498, -1.396635, -2.557937, -0.757816, 1.570796, 1.934294],accel_mss,speed_ms,0,blend_radius_m)
      movel([0.362999, -1.396660, -2.557920, -0.757810, 1.570796, 1.933796],accel_mss,speed_ms,0,blend_radius_m)
      movel([0.362504, -1.396675, -2.557908, -0.757805, 1.570796, 1.933301],accel_mss,speed_ms,0,blend_radius_m)
      movel([0.362015, -1.396682, -2.557903, -0.757803, 1.570796, 1.932811],accel_mss,speed_ms,0,blend_radius_m)
      movel([0.361806, -1.396678, -2.557906, -0.757805, 1.570796, 1.932602],accel_mss,speed_ms,0,blend_radius_m)
      movel([0.361605, -1.396664, -2.557916, -0.757808, 1.570796, 1.932402],accel_mss,speed_ms,0,blend_radius_m)
      movel([0.361406, -1.396642, -2.557932, -0.757814, 1.570796, 1.932202],accel_mss,speed_ms,0,blend_radius_m)
      movel([0.361238, -1.396615, -2.557953, -0.757822, 1.570796, 1.932034],accel_mss,speed_ms,0,blend_radius_m)
      movel([0.361077, -1.396576, -2.557981, -0.757832, 1.570796, 1.931873],accel_mss,speed_ms,0,blend_radius_m)
      movel([0.360921, -1.396528, -2.558016, -0.757845, 1.570796, 1.931717],accel_mss,speed_ms,0,blend_radius_m)
      movel([0.360646, -1.396422, -2.558093, -0.757874, 1.570796, 1.931442],accel_mss,speed_ms,0,blend_radius_m)
      movel([0.360383, -1.396300, -2.558182, -0.757907, 1.570796, 1.931179],accel_mss,speed_ms,0,blend_radius_m)
      movel([0.360162, -1.396184, -2.558267, -0.757938, 1.570796, 1.930958],accel_mss,speed_ms,0,blend_radius_m)
      movel([0.359955, -1.396051, -2.558364, -0.757974, 1.570796, 1.930752],accel_mss,speed_ms,0,blend_radius_m)
      movel([0.359760, -1.395907, -2.558468, -0.758013, 1.570796, 1.930556],accel_mss,speed_ms,0,blend_radius_m)
      movel([0.359578, -1.395752, -2.558582, -0.758056, 1.570796, 1.930375],accel_mss,speed_ms,0,blend_radius_m)
      movel([0.359396, -1.395570, -2.558714, -0.758105, 1.570796, 1.930192],accel_mss,speed_ms,0,blend_radius_m)
      movel([0.359225, -1.395380, -2.558853, -0.758157, 1.570796, 1.930022],accel_mss,speed_ms,0,blend_radius_m)
      movel([0.359065, -1.395180, -2.558998, -0.758211, 1.570796, 1.929862],accel_mss,speed_ms,0,blend_radius_m)
      movel([0.358920, -1.394971, -2.559150, -0.758268, 1.570796, 1.929717],accel_mss,speed_ms,0,blend_radius_m)
      movel([0.358783, -1.394746, -2.559314, -0.758330, 1.570796, 1.929580],accel_mss,speed_ms,0,blend_radius_m)
      movel([0.358658, -1.394514, -2.559482, -0.758393, 1.570796, 1.929455],accel_mss,speed_ms,0,blend_radius_m)
      movel([0.358548, -1.394272, -2.559658, -0.758459, 1.570796, 1.929345],accel_mss,speed_ms,0,blend_radius_m)
      movel([0.358450, -1.394024, -2.559838, -0.758527, 1.570796, 1.929246],accel_mss,speed_ms,0,blend_radius_m)
      movel([0.358370, -1.393774, -2.560019, -0.758596, 1.570796, 1.929166],accel_mss,speed_ms,0,blend_radius_m)
      movel([0.358304, -1.393517, -2.560206, -0.758666, 1.570796, 1.929101],accel_mss,speed_ms,0,blend_radius_m)
      movel([0.358253, -1.393253, -2.560397, -0.758739, 1.570796, 1.929049],accel_mss,speed_ms,0,blend_radius_m)
      movel([0.358218, -1.392982, -2.560594, -0.758814, 1.570796, 1.929014],accel_mss,speed_ms,0,blend_radius_m)
      movel([0.358185, -1.392609, -2.560863, -0.758916, 1.570796, 1.928982],accel_mss,speed_ms,0,blend_radius_m)
      movel([0.358172, -1.392230, -2.561138, -0.759021, 1.570796, 1.928968],accel_mss,speed_ms,0,blend_radius_m)
      movel([0.358176, -1.392048, -2.561270, -0.759072, 1.570796, 1.928973],accel_mss,speed_ms,0,blend_radius_m)
      movel([0.358197, -1.391861, -2.561405, -0.759123, 1.570796, 1.928993],accel_mss,speed_ms,0,blend_radius_m)
      movel([0.358230, -1.391671, -2.561542, -0.759176, 1.570796, 1.929026],accel_mss,speed_ms,0,blend_radius_m)
      movel([0.358284, -1.391445, -2.561705, -0.759239, 1.570796, 1.929080],accel_mss,speed_ms,0,blend_radius_m)
      movel([0.358349, -1.391219, -2.561868, -0.759302, 1.570796, 1.929145],accel_mss,speed_ms,0,blend_radius_m)
      movel([0.358426, -1.390992, -2.562032, -0.759365, 1.570796, 1.929222],accel_mss,speed_ms,0,blend_radius_m)
      speed_ms = 0.003
      movel([0.358426, -1.394245, -2.563502, -0.754642, 1.570796, 1.929222],accel_mss,speed_ms,0,blend_radius_m)
      speed_ms = 0.007
      movel([0.358674, -1.393582, -2.563983, -0.754824, 1.570796, 1.929470],accel_mss,speed_ms,0,blend_radius_m)
      movel([0.358928, -1.392920, -2.564462, -0.755007, 1.570796, 1.929724],accel_mss,speed_ms,0,blend_radius_m)
      movel([0.359196, -1.392246, -2.564949, -0.755194, 1.570796, 1.929992],accel_mss,speed_ms,0,blend_radius_m)
      movel([0.359471, -1.391570, -2.565436, -0.755382, 1.570796, 1.930267],accel_mss,speed_ms,0,blend_radius_m)
      movel([0.359570, -1.391346, -2.565598, -0.755445, 1.570796, 1.930367],accel_mss,speed_ms,0,blend_radius_m)
      movel([0.359681, -1.391122, -2.565760, -0.755507, 1.570796, 1.930477],accel_mss,speed_ms,0,blend_radius_m)
      movel([0.359803, -1.390898, -2.565921, -0.755570, 1.570796, 1.930599],accel_mss,speed_ms,0,blend_radius_m)
      movel([0.359919, -1.390706, -2.566059, -0.755624, 1.570796, 1.930715],accel_mss,speed_ms,0,blend_radius_m)
      movel([0.360048, -1.390518, -2.566195, -0.755676, 1.570796, 1.930844],accel_mss,speed_ms,0,blend_radius_m)
      movel([0.360189, -1.390333, -2.566328, -0.755728, 1.570796, 1.930985],accel_mss,speed_ms,0,blend_radius_m)
      movel([0.360518, -1.389930, -2.566617, -0.755841, 1.570796, 1.931314],accel_mss,speed_ms,0,blend_radius_m)
      movel([0.360858, -1.389536, -2.566901, -0.755952, 1.570796, 1.931654],accel_mss,speed_ms,0,blend_radius_m)
      movel([0.361119, -1.389248, -2.567107, -0.756034, 1.570796, 1.931916],accel_mss,speed_ms,0,blend_radius_m)
      movel([0.361388, -1.388967, -2.567309, -0.756113, 1.570796, 1.932184],accel_mss,speed_ms,0,blend_radius_m)
      movel([0.361665, -1.388692, -2.567506, -0.756191, 1.570796, 1.932462],accel_mss,speed_ms,0,blend_radius_m)
      movel([0.361951, -1.388421, -2.567701, -0.756268, 1.570796, 1.932747],accel_mss,speed_ms,0,blend_radius_m)
      movel([0.362243, -1.388160, -2.567888, -0.756342, 1.570796, 1.933040],accel_mss,speed_ms,0,blend_radius_m)
      movel([0.362544, -1.387903, -2.568071, -0.756414, 1.570796, 1.933340],accel_mss,speed_ms,0,blend_radius_m)
      movel([0.362850, -1.387655, -2.568249, -0.756485, 1.570796, 1.933646],accel_mss,speed_ms,0,blend_radius_m)
      movel([0.363162, -1.387415, -2.568420, -0.756553, 1.570796, 1.933959],accel_mss,speed_ms,0,blend_radius_m)
      movel([0.363474, -1.387189, -2.568582, -0.756618, 1.570796, 1.934270],accel_mss,speed_ms,0,blend_radius_m)
      movel([0.363789, -1.386971, -2.568738, -0.756680, 1.570796, 1.934586],accel_mss,speed_ms,0,blend_radius_m)
      movel([0.364110, -1.386764, -2.568886, -0.756739, 1.570796, 1.934906],accel_mss,speed_ms,0,blend_radius_m)
      movel([0.364437, -1.386564, -2.569029, -0.756796, 1.570796, 1.935233],accel_mss,speed_ms,0,blend_radius_m)
      movel([0.364752, -1.386384, -2.569158, -0.756848, 1.570796, 1.935548],accel_mss,speed_ms,0,blend_radius_m)
      movel([0.365072, -1.386212, -2.569280, -0.756897, 1.570796, 1.935868],accel_mss,speed_ms,0,blend_radius_m)
      movel([0.365394, -1.386054, -2.569393, -0.756942, 1.570796, 1.936190],accel_mss,speed_ms,0,blend_radius_m)
      movel([0.365717, -1.385907, -2.569498, -0.756985, 1.570796, 1.936513],accel_mss,speed_ms,0,blend_radius_m)
      movel([0.366119, -1.385738, -2.569618, -0.757033, 1.570796, 1.936915],accel_mss,speed_ms,0,blend_radius_m)
      movel([0.366520, -1.385583, -2.569728, -0.757077, 1.570796, 1.937316],accel_mss,speed_ms,0,blend_radius_m)
      movel([0.366722, -1.385515, -2.569777, -0.757097, 1.570796, 1.937518],accel_mss,speed_ms,0,blend_radius_m)
      movel([0.366925, -1.385455, -2.569820, -0.757114, 1.570796, 1.937721],accel_mss,speed_ms,0,blend_radius_m)
      movel([0.367125, -1.385409, -2.569853, -0.757128, 1.570796, 1.937921],accel_mss,speed_ms,0,blend_radius_m)
      movel([0.367346, -1.385366, -2.569883, -0.757140, 1.570796, 1.938143],accel_mss,speed_ms,0,blend_radius_m)
      movel([0.367566, -1.385335, -2.569905, -0.757149, 1.570796, 1.938362],accel_mss,speed_ms,0,blend_radius_m)
      movel([0.367783, -1.385314, -2.569920, -0.757155, 1.570796, 1.938579],accel_mss,speed_ms,0,blend_radius_m)
      movel([0.368308, -1.385277, -2.569947, -0.757166, 1.570796, 1.939104],accel_mss,speed_ms,0,blend_radius_m)
      movel([0.368831, -1.385251, -2.569965, -0.757173, 1.570796, 1.939627],accel_mss,speed_ms,0,blend_radius_m)
      movel([0.369362, -1.385234, -2.569977, -0.757178, 1.570796, 1.940158],accel_mss,speed_ms,0,blend_radius_m)
      movel([0.369888, -1.385228, -2.569981, -0.757180, 1.570796, 1.940684],accel_mss,speed_ms,0,blend_radius_m)
      movel([0.370095, -1.385233, -2.569978, -0.757178, 1.570796, 1.940891],accel_mss,speed_ms,0,blend_radius_m)
      movel([0.370296, -1.385247, -2.569968, -0.757174, 1.570796, 1.941092],accel_mss,speed_ms,0,blend_radius_m)
      movel([0.370489, -1.385275, -2.569948, -0.757166, 1.570796, 1.941285],accel_mss,speed_ms,0,blend_radius_m)
      movel([0.370661, -1.385311, -2.569922, -0.757156, 1.570796, 1.941457],accel_mss,speed_ms,0,blend_radius_m)
      movel([0.370825, -1.385360, -2.569887, -0.757142, 1.570796, 1.941621],accel_mss,speed_ms,0,blend_radius_m)
      movel([0.370983, -1.385418, -2.569846, -0.757125, 1.570796, 1.941779],accel_mss,speed_ms,0,blend_radius_m)
      movel([0.371305, -1.385566, -2.569741, -0.757083, 1.570796, 1.942101],accel_mss,speed_ms,0,blend_radius_m)
      movel([0.371615, -1.385725, -2.569627, -0.757037, 1.570796, 1.942412],accel_mss,speed_ms,0,blend_radius_m)
      movel([0.371844, -1.385858, -2.569532, -0.756998, 1.570796, 1.942640],accel_mss,speed_ms,0,blend_radius_m)
      movel([0.372062, -1.386006, -2.569427, -0.756956, 1.570796, 1.942859],accel_mss,speed_ms,0,blend_radius_m)
      movel([0.372266, -1.386167, -2.569312, -0.756910, 1.570796, 1.943062],accel_mss,speed_ms,0,blend_radius_m)
      movel([0.372459, -1.386337, -2.569190, -0.756861, 1.570796, 1.943255],accel_mss,speed_ms,0,blend_radius_m)
      movel([0.372637, -1.386522, -2.569059, -0.756808, 1.570796, 1.943433],accel_mss,speed_ms,0,blend_radius_m)
      movel([0.372801, -1.386718, -2.568919, -0.756752, 1.570796, 1.943597],accel_mss,speed_ms,0,blend_radius_m)
      movel([0.372948, -1.386926, -2.568770, -0.756693, 1.570796, 1.943745],accel_mss,speed_ms,0,blend_radius_m)
      movel([0.373083, -1.387143, -2.568615, -0.756631, 1.570796, 1.943879],accel_mss,speed_ms,0,blend_radius_m)
      movel([0.373225, -1.387411, -2.568424, -0.756554, 1.570796, 1.944021],accel_mss,speed_ms,0,blend_radius_m)
      movel([0.373345, -1.387690, -2.568224, -0.756475, 1.570796, 1.944142],accel_mss,speed_ms,0,blend_radius_m)
      movel([0.373450, -1.387982, -2.568015, -0.756392, 1.570796, 1.944246],accel_mss,speed_ms,0,blend_radius_m)
      movel([0.373533, -1.388285, -2.567798, -0.756306, 1.570796, 1.944329],accel_mss,speed_ms,0,blend_radius_m)
      movel([0.373597, -1.388597, -2.567574, -0.756218, 1.570796, 1.944393],accel_mss,speed_ms,0,blend_radius_m)
      movel([0.373641, -1.388917, -2.567345, -0.756127, 1.570796, 1.944437],accel_mss,speed_ms,0,blend_radius_m)
      movel([0.373668, -1.389246, -2.567109, -0.756034, 1.570796, 1.944464],accel_mss,speed_ms,0,blend_radius_m)
      movel([0.373674, -1.389586, -2.566864, -0.755938, 1.570796, 1.944470],accel_mss,speed_ms,0,blend_radius_m)
      movel([0.373659, -1.389934, -2.566615, -0.755840, 1.570796, 1.944455],accel_mss,speed_ms,0,blend_radius_m)
      movel([0.373627, -1.390289, -2.566359, -0.755741, 1.570796, 1.944423],accel_mss,speed_ms,0,blend_radius_m)
      movel([0.373576, -1.390647, -2.566102, -0.755640, 1.570796, 1.944372],accel_mss,speed_ms,0,blend_radius_m)
      movel([0.373503, -1.391011, -2.565839, -0.755538, 1.570796, 1.944300],accel_mss,speed_ms,0,blend_radius_m)
      movel([0.373412, -1.391376, -2.565576, -0.755436, 1.570796, 1.944209],accel_mss,speed_ms,0,blend_radius_m)
      movel([0.373304, -1.391746, -2.565310, -0.755333, 1.570796, 1.944100],accel_mss,speed_ms,0,blend_radius_m)
      movel([0.373175, -1.392114, -2.565044, -0.755231, 1.570796, 1.943971],accel_mss,speed_ms,0,blend_radius_m)
      movel([0.373030, -1.392483, -2.564778, -0.755128, 1.570796, 1.943827],accel_mss,speed_ms,0,blend_radius_m)
      movel([0.372866, -1.392854, -2.564509, -0.755025, 1.570796, 1.943663],accel_mss,speed_ms,0,blend_radius_m)
      movel([0.372686, -1.393221, -2.564244, -0.754924, 1.570796, 1.943482],accel_mss,speed_ms,0,blend_radius_m)
      movel([0.372487, -1.393589, -2.563978, -0.754822, 1.570796, 1.943283],accel_mss,speed_ms,0,blend_radius_m)
      movel([0.372271, -1.393954, -2.563713, -0.754722, 1.570796, 1.943067],accel_mss,speed_ms,0,blend_radius_m)
      movel([0.372039, -1.394314, -2.563452, -0.754623, 1.570796, 1.942835],accel_mss,speed_ms,0,blend_radius_m)
      movel([0.371814, -1.394638, -2.563217, -0.754534, 1.570796, 1.942611],accel_mss,speed_ms,0,blend_radius_m)
      movel([0.371581, -1.394957, -2.562985, -0.754446, 1.570796, 1.942377],accel_mss,speed_ms,0,blend_radius_m)
      movel([0.371333, -1.395273, -2.562756, -0.754360, 1.570796, 1.942129],accel_mss,speed_ms,0,blend_radius_m)
      movel([0.371076, -1.395582, -2.562532, -0.754275, 1.570796, 1.941872],accel_mss,speed_ms,0,blend_radius_m)
      movel([0.370810, -1.395887, -2.562310, -0.754192, 1.570796, 1.941606],accel_mss,speed_ms,0,blend_radius_m)
      movel([0.370537, -1.396181, -2.562096, -0.754112, 1.570796, 1.941333],accel_mss,speed_ms,0,blend_radius_m)
      movel([0.370253, -1.396467, -2.561888, -0.754034, 1.570796, 1.941050],accel_mss,speed_ms,0,blend_radius_m)
      movel([0.369963, -1.396744, -2.561686, -0.753959, 1.570796, 1.940759],accel_mss,speed_ms,0,blend_radius_m)
      movel([0.369663, -1.397015, -2.561488, -0.753886, 1.570796, 1.940459],accel_mss,speed_ms,0,blend_radius_m)
      movel([0.369355, -1.397277, -2.561297, -0.753815, 1.570796, 1.940152],accel_mss,speed_ms,0,blend_radius_m)
      movel([0.369041, -1.397528, -2.561114, -0.753747, 1.570796, 1.939837],accel_mss,speed_ms,0,blend_radius_m)
      movel([0.368722, -1.397769, -2.560938, -0.753682, 1.570796, 1.939518],accel_mss,speed_ms,0,blend_radius_m)
      movel([0.368395, -1.398001, -2.560769, -0.753619, 1.570796, 1.939192],accel_mss,speed_ms,0,blend_radius_m)
      movel([0.368064, -1.398222, -2.560607, -0.753560, 1.570796, 1.938860],accel_mss,speed_ms,0,blend_radius_m)
      movel([0.367728, -1.398433, -2.560453, -0.753503, 1.570796, 1.938524],accel_mss,speed_ms,0,blend_radius_m)
      movel([0.367387, -1.398633, -2.560307, -0.753450, 1.570796, 1.938184],accel_mss,speed_ms,0,blend_radius_m)
      movel([0.367040, -1.398822, -2.560168, -0.753399, 1.570796, 1.937836],accel_mss,speed_ms,0,blend_radius_m)
      movel([0.366693, -1.398998, -2.560039, -0.753351, 1.570796, 1.937489],accel_mss,speed_ms,0,blend_radius_m)
      movel([0.366341, -1.399164, -2.559918, -0.753307, 1.570796, 1.937138],accel_mss,speed_ms,0,blend_radius_m)
      movel([0.365988, -1.399316, -2.559806, -0.753266, 1.570796, 1.936785],accel_mss,speed_ms,0,blend_radius_m)
      movel([0.365621, -1.399461, -2.559701, -0.753228, 1.570796, 1.936417],accel_mss,speed_ms,0,blend_radius_m)
      movel([0.365251, -1.399592, -2.559604, -0.753193, 1.570796, 1.936047],accel_mss,speed_ms,0,blend_radius_m)
      movel([0.365052, -1.399654, -2.559559, -0.753176, 1.570796, 1.935848],accel_mss,speed_ms,0,blend_radius_m)
      movel([0.364854, -1.399707, -2.559520, -0.753162, 1.570796, 1.935651],accel_mss,speed_ms,0,blend_radius_m)
      movel([0.364658, -1.399752, -2.559487, -0.753150, 1.570796, 1.935454],accel_mss,speed_ms,0,blend_radius_m)
      movel([0.364437, -1.399789, -2.559460, -0.753140, 1.570796, 1.935233],accel_mss,speed_ms,0,blend_radius_m)
      movel([0.364217, -1.399819, -2.559438, -0.753132, 1.570796, 1.935013],accel_mss,speed_ms,0,blend_radius_m)
      movel([0.364000, -1.399841, -2.559422, -0.753126, 1.570796, 1.934796],accel_mss,speed_ms,0,blend_radius_m)
      movel([0.363498, -1.399873, -2.559398, -0.753118, 1.570796, 1.934294],accel_mss,speed_ms,0,blend_radius_m)
      movel([0.362999, -1.399898, -2.559380, -0.753111, 1.570796, 1.933796],accel_mss,speed_ms,0,blend_radius_m)
      movel([0.362504, -1.399913, -2.559369, -0.753107, 1.570796, 1.933301],accel_mss,speed_ms,0,blend_radius_m)
      movel([0.362015, -1.399920, -2.559364, -0.753105, 1.570796, 1.932811],accel_mss,speed_ms,0,blend_radius_m)
      movel([0.361806, -1.399916, -2.559367, -0.753106, 1.570796, 1.932602],accel_mss,speed_ms,0,blend_radius_m)
      movel([0.361605, -1.399902, -2.559377, -0.753110, 1.570796, 1.932402],accel_mss,speed_ms,0,blend_radius_m)
      movel([0.361406, -1.399880, -2.559393, -0.753116, 1.570796, 1.932202],accel_mss,speed_ms,0,blend_radius_m)
      movel([0.361238, -1.399853, -2.559413, -0.753123, 1.570796, 1.932034],accel_mss,speed_ms,0,blend_radius_m)
      movel([0.361077, -1.399814, -2.559442, -0.753133, 1.570796, 1.931873],accel_mss,speed_ms,0,blend_radius_m)
      movel([0.360921, -1.399766, -2.559477, -0.753146, 1.570796, 1.931717],accel_mss,speed_ms,0,blend_radius_m)
      movel([0.360646, -1.399661, -2.559554, -0.753174, 1.570796, 1.931442],accel_mss,speed_ms,0,blend_radius_m)
      movel([0.360383, -1.399539, -2.559643, -0.753207, 1.570796, 1.931179],accel_mss,speed_ms,0,blend_radius_m)
      movel([0.360162, -1.399423, -2.559728, -0.753238, 1.570796, 1.930958],accel_mss,speed_ms,0,blend_radius_m)
      movel([0.359955, -1.399291, -2.559825, -0.753273, 1.570796, 1.930752],accel_mss,speed_ms,0,blend_radius_m)
      movel([0.359760, -1.399147, -2.559930, -0.753312, 1.570796, 1.930556],accel_mss,speed_ms,0,blend_radius_m)
      movel([0.359578, -1.398992, -2.560044, -0.753353, 1.570796, 1.930375],accel_mss,speed_ms,0,blend_radius_m)
      movel([0.359396, -1.398811, -2.560176, -0.753402, 1.570796, 1.930192],accel_mss,speed_ms,0,blend_radius_m)
      movel([0.359225, -1.398621, -2.560315, -0.753453, 1.570796, 1.930022],accel_mss,speed_ms,0,blend_radius_m)
      movel([0.359065, -1.398422, -2.560461, -0.753506, 1.570796, 1.929862],accel_mss,speed_ms,0,blend_radius_m)
      movel([0.358920, -1.398213, -2.560613, -0.753562, 1.570796, 1.929717],accel_mss,speed_ms,0,blend_radius_m)
      movel([0.358783, -1.397989, -2.560777, -0.753623, 1.570796, 1.929580],accel_mss,speed_ms,0,blend_radius_m)
      movel([0.358658, -1.397758, -2.560946, -0.753685, 1.570796, 1.929455],accel_mss,speed_ms,0,blend_radius_m)
      movel([0.358548, -1.397517, -2.561122, -0.753750, 1.570796, 1.929345],accel_mss,speed_ms,0,blend_radius_m)
      movel([0.358450, -1.397269, -2.561303, -0.753817, 1.570796, 1.929246],accel_mss,speed_ms,0,blend_radius_m)
      movel([0.358370, -1.397020, -2.561485, -0.753884, 1.570796, 1.929166],accel_mss,speed_ms,0,blend_radius_m)
      movel([0.358304, -1.396764, -2.561671, -0.753954, 1.570796, 1.929101],accel_mss,speed_ms,0,blend_radius_m)
      movel([0.358253, -1.396501, -2.561863, -0.754025, 1.570796, 1.929049],accel_mss,speed_ms,0,blend_radius_m)
      movel([0.358218, -1.396230, -2.562060, -0.754099, 1.570796, 1.929014],accel_mss,speed_ms,0,blend_radius_m)
      movel([0.358185, -1.395859, -2.562330, -0.754200, 1.570796, 1.928982],accel_mss,speed_ms,0,blend_radius_m)
      movel([0.358172, -1.395480, -2.562606, -0.754303, 1.570796, 1.928968],accel_mss,speed_ms,0,blend_radius_m)
      movel([0.358176, -1.395299, -2.562738, -0.754353, 1.570796, 1.928973],accel_mss,speed_ms,0,blend_radius_m)
      movel([0.358197, -1.395112, -2.562873, -0.754404, 1.570796, 1.928993],accel_mss,speed_ms,0,blend_radius_m)
      movel([0.358230, -1.394923, -2.563010, -0.754456, 1.570796, 1.929026],accel_mss,speed_ms,0,blend_radius_m)
      movel([0.358284, -1.394698, -2.563174, -0.754517, 1.570796, 1.929080],accel_mss,speed_ms,0,blend_radius_m)
      movel([0.358349, -1.394472, -2.563338, -0.754579, 1.570796, 1.929145],accel_mss,speed_ms,0,blend_radius_m)
      movel([0.358426, -1.394245, -2.563502, -0.754642, 1.570796, 1.929222],accel_mss,speed_ms,0,blend_radius_m)
      speed_ms = 0.003
      movel([0.358426, -1.381362, -2.557573, -0.773455, 1.570796, 1.929222],accel_mss,speed_ms,0,blend_radius_m)
      speed_ms = 0.01
      movel([0.358426, -1.356634, -2.545321, -0.810434, 1.570796, 1.929222],accel_mss,speed_ms,0,blend_radius_m)
      movel([0.346697, -1.391181, -2.520822, -0.800386, 1.570796, 1.917493],accel_mss,speed_ms,0,blend_radius_m)
      movel([0.346697, -1.415265, -2.532641, -0.764483, 1.570796, 1.917493],accel_mss,speed_ms,0,blend_radius_m)
      speed_ms = 0.003
      movel([0.346697, -1.424623, -2.536939, -0.750828, 1.570796, 1.917493],accel_mss,speed_ms,0,blend_radius_m)
      speed_ms = 0.007
      movel([0.346787, -1.424640, -2.536926, -0.750824, 1.570796, 1.917583],accel_mss,speed_ms,0,blend_radius_m)
      movel([0.346871, -1.424667, -2.536904, -0.750817, 1.570796, 1.917667],accel_mss,speed_ms,0,blend_radius_m)
      movel([0.346947, -1.424703, -2.536876, -0.750809, 1.570796, 1.917744],accel_mss,speed_ms,0,blend_radius_m)
      movel([0.347017, -1.424746, -2.536843, -0.750799, 1.570796, 1.917813],accel_mss,speed_ms,0,blend_radius_m)
      movel([0.347080, -1.424806, -2.536797, -0.750786, 1.570796, 1.917876],accel_mss,speed_ms,0,blend_radius_m)
      movel([0.347134, -1.424872, -2.536746, -0.750770, 1.570796, 1.917930],accel_mss,speed_ms,0,blend_radius_m)
      movel([0.347175, -1.424948, -2.536688, -0.750753, 1.570796, 1.917971],accel_mss,speed_ms,0,blend_radius_m)
      movel([0.347205, -1.425032, -2.536623, -0.750734, 1.570796, 1.918001],accel_mss,speed_ms,0,blend_radius_m)
      movel([0.347218, -1.425123, -2.536553, -0.750713, 1.570796, 1.918014],accel_mss,speed_ms,0,blend_radius_m)
      movel([0.347222, -1.425216, -2.536481, -0.750692, 1.570796, 1.918018],accel_mss,speed_ms,0,blend_radius_m)
      movel([0.347208, -1.425340, -2.536385, -0.750664, 1.570796, 1.918004],accel_mss,speed_ms,0,blend_radius_m)
      movel([0.347175, -1.425466, -2.536288, -0.750635, 1.570796, 1.917971],accel_mss,speed_ms,0,blend_radius_m)
      movel([0.347126, -1.425593, -2.536190, -0.750606, 1.570796, 1.917923],accel_mss,speed_ms,0,blend_radius_m)
      movel([0.347060, -1.425721, -2.536091, -0.750577, 1.570796, 1.917856],accel_mss,speed_ms,0,blend_radius_m)
      movel([0.346979, -1.425847, -2.535994, -0.750548, 1.570796, 1.917775],accel_mss,speed_ms,0,blend_radius_m)
      movel([0.346883, -1.425965, -2.535902, -0.750522, 1.570796, 1.917679],accel_mss,speed_ms,0,blend_radius_m)
      movel([0.346776, -1.426078, -2.535815, -0.750496, 1.570796, 1.917573],accel_mss,speed_ms,0,blend_radius_m)
      movel([0.346658, -1.426181, -2.535735, -0.750473, 1.570796, 1.917454],accel_mss,speed_ms,0,blend_radius_m)
      movel([0.346533, -1.426273, -2.535664, -0.750452, 1.570796, 1.917329],accel_mss,speed_ms,0,blend_radius_m)
      movel([0.346398, -1.426356, -2.535600, -0.750433, 1.570796, 1.917194],accel_mss,speed_ms,0,blend_radius_m)
      movel([0.346286, -1.426413, -2.535556, -0.750420, 1.570796, 1.917083],accel_mss,speed_ms,0,blend_radius_m)
      movel([0.346173, -1.426457, -2.535521, -0.750410, 1.570796, 1.916969],accel_mss,speed_ms,0,blend_radius_m)
      movel([0.346061, -1.426491, -2.535495, -0.750402, 1.570796, 1.916857],accel_mss,speed_ms,0,blend_radius_m)
      movel([0.345947, -1.426515, -2.535477, -0.750397, 1.570796, 1.916743],accel_mss,speed_ms,0,blend_radius_m)
      movel([0.345839, -1.426526, -2.535468, -0.750395, 1.570796, 1.916636],accel_mss,speed_ms,0,blend_radius_m)
      movel([0.345734, -1.426526, -2.535468, -0.750395, 1.570796, 1.916530],accel_mss,speed_ms,0,blend_radius_m)
      movel([0.345634, -1.426512, -2.535479, -0.750398, 1.570796, 1.916430],accel_mss,speed_ms,0,blend_radius_m)
      movel([0.345544, -1.426483, -2.535502, -0.750404, 1.570796, 1.916340],accel_mss,speed_ms,0,blend_radius_m)
      movel([0.345462, -1.426443, -2.535533, -0.750413, 1.570796, 1.916259],accel_mss,speed_ms,0,blend_radius_m)
      movel([0.345395, -1.426390, -2.535574, -0.750425, 1.570796, 1.916191],accel_mss,speed_ms,0,blend_radius_m)
      movel([0.345334, -1.426320, -2.535628, -0.750441, 1.570796, 1.916130],accel_mss,speed_ms,0,blend_radius_m)
      movel([0.345282, -1.426241, -2.535689, -0.750459, 1.570796, 1.916079],accel_mss,speed_ms,0,blend_radius_m)
      movel([0.345245, -1.426155, -2.535755, -0.750479, 1.570796, 1.916041],accel_mss,speed_ms,0,blend_radius_m)
      movel([0.345220, -1.426063, -2.535827, -0.750499, 1.570796, 1.916017],accel_mss,speed_ms,0,blend_radius_m)
      movel([0.345208, -1.425964, -2.535903, -0.750522, 1.570796, 1.916004],accel_mss,speed_ms,0,blend_radius_m)
      movel([0.345210, -1.425860, -2.535984, -0.750546, 1.570796, 1.916006],accel_mss,speed_ms,0,blend_radius_m)
      movel([0.345225, -1.425751, -2.536068, -0.750570, 1.570796, 1.916021],accel_mss,speed_ms,0,blend_radius_m)
      movel([0.345253, -1.425641, -2.536152, -0.750595, 1.570796, 1.916049],accel_mss,speed_ms,0,blend_radius_m)
      movel([0.345292, -1.425540, -2.536231, -0.750618, 1.570796, 1.916088],accel_mss,speed_ms,0,blend_radius_m)
      movel([0.345346, -1.425438, -2.536310, -0.750642, 1.570796, 1.916142],accel_mss,speed_ms,0,blend_radius_m)
      movel([0.345412, -1.425339, -2.536386, -0.750664, 1.570796, 1.916208],accel_mss,speed_ms,0,blend_radius_m)
      movel([0.345491, -1.425246, -2.536458, -0.750685, 1.570796, 1.916288],accel_mss,speed_ms,0,blend_radius_m)
      movel([0.345618, -1.425116, -2.536558, -0.750715, 1.570796, 1.916414],accel_mss,speed_ms,0,blend_radius_m)
      movel([0.345757, -1.424993, -2.536653, -0.750743, 1.570796, 1.916553],accel_mss,speed_ms,0,blend_radius_m)
      movel([0.345901, -1.424880, -2.536740, -0.750769, 1.570796, 1.916697],accel_mss,speed_ms,0,blend_radius_m)
      movel([0.346001, -1.424814, -2.536791, -0.750784, 1.570796, 1.916798],accel_mss,speed_ms,0,blend_radius_m)
      movel([0.346103, -1.424755, -2.536837, -0.750797, 1.570796, 1.916899],accel_mss,speed_ms,0,blend_radius_m)
      movel([0.346209, -1.424707, -2.536874, -0.750808, 1.570796, 1.917006],accel_mss,speed_ms,0,blend_radius_m)
      movel([0.346315, -1.424666, -2.536905, -0.750818, 1.570796, 1.917111],accel_mss,speed_ms,0,blend_radius_m)
      movel([0.346415, -1.424639, -2.536926, -0.750824, 1.570796, 1.917212],accel_mss,speed_ms,0,blend_radius_m)
      movel([0.346512, -1.424622, -2.536939, -0.750828, 1.570796, 1.917308],accel_mss,speed_ms,0,blend_radius_m)
      movel([0.346606, -1.424618, -2.536942, -0.750829, 1.570796, 1.917402],accel_mss,speed_ms,0,blend_radius_m)
      movel([0.346697, -1.424623, -2.536939, -0.750828, 1.570796, 1.917493],accel_mss,speed_ms,0,blend_radius_m)
      speed_ms = 0.003
      movel([0.346697, -1.427782, -2.538354, -0.746253, 1.570796, 1.917493],accel_mss,speed_ms,0,blend_radius_m)
      speed_ms = 0.007
      movel([0.346787, -1.427799, -2.538341, -0.746249, 1.570796, 1.917583],accel_mss,speed_ms,0,blend_radius_m)
      movel([0.346871, -1.427826, -2.538320, -0.746243, 1.570796, 1.917667],accel_mss,speed_ms,0,blend_radius_m)
      movel([0.346947, -1.427862, -2.538292, -0.746235, 1.570796, 1.917744],accel_mss,speed_ms,0,blend_radius_m)
      movel([0.347017, -1.427905, -2.538259, -0.746225, 1.570796, 1.917813],accel_mss,speed_ms,0,blend_radius_m)
      movel([0.347080, -1.427965, -2.538213, -0.746212, 1.570796, 1.917876],accel_mss,speed_ms,0,blend_radius_m)
      movel([0.347134, -1.428031, -2.538161, -0.746197, 1.570796, 1.917930],accel_mss,speed_ms,0,blend_radius_m)
      movel([0.347175, -1.428106, -2.538103, -0.746180, 1.570796, 1.917971],accel_mss,speed_ms,0,blend_radius_m)
      movel([0.347205, -1.428190, -2.538038, -0.746161, 1.570796, 1.918001],accel_mss,speed_ms,0,blend_radius_m)
      movel([0.347218, -1.428281, -2.537968, -0.746141, 1.570796, 1.918014],accel_mss,speed_ms,0,blend_radius_m)
      movel([0.347222, -1.428374, -2.537895, -0.746120, 1.570796, 1.918018],accel_mss,speed_ms,0,blend_radius_m)
      movel([0.347208, -1.428497, -2.537800, -0.746092, 1.570796, 1.918004],accel_mss,speed_ms,0,blend_radius_m)
      movel([0.347175, -1.428623, -2.537702, -0.746064, 1.570796, 1.917971],accel_mss,speed_ms,0,blend_radius_m)
      movel([0.347126, -1.428749, -2.537604, -0.746036, 1.570796, 1.917923],accel_mss,speed_ms,0,blend_radius_m)
      movel([0.347060, -1.428877, -2.537505, -0.746007, 1.570796, 1.917856],accel_mss,speed_ms,0,blend_radius_m)
      movel([0.346979, -1.429002, -2.537407, -0.745979, 1.570796, 1.917775],accel_mss,speed_ms,0,blend_radius_m)
      movel([0.346883, -1.429121, -2.537316, -0.745953, 1.570796, 1.917679],accel_mss,speed_ms,0,blend_radius_m)
      movel([0.346776, -1.429233, -2.537228, -0.745928, 1.570796, 1.917573],accel_mss,speed_ms,0,blend_radius_m)
      movel([0.346658, -1.429335, -2.537149, -0.745905, 1.570796, 1.917454],accel_mss,speed_ms,0,blend_radius_m)
      movel([0.346533, -1.429428, -2.537077, -0.745884, 1.570796, 1.917329],accel_mss,speed_ms,0,blend_radius_m)
      movel([0.346398, -1.429510, -2.537013, -0.745866, 1.570796, 1.917194],accel_mss,speed_ms,0,blend_radius_m)
      movel([0.346286, -1.429567, -2.536969, -0.745853, 1.570796, 1.917083],accel_mss,speed_ms,0,blend_radius_m)
      movel([0.346173, -1.429611, -2.536934, -0.745843, 1.570796, 1.916969],accel_mss,speed_ms,0,blend_radius_m)
      movel([0.346061, -1.429645, -2.536908, -0.745836, 1.570796, 1.916857],accel_mss,speed_ms,0,blend_radius_m)
      movel([0.345947, -1.429669, -2.536890, -0.745831, 1.570796, 1.916743],accel_mss,speed_ms,0,blend_radius_m)
      movel([0.345839, -1.429679, -2.536881, -0.745828, 1.570796, 1.916636],accel_mss,speed_ms,0,blend_radius_m)
      movel([0.345734, -1.429680, -2.536881, -0.745828, 1.570796, 1.916530],accel_mss,speed_ms,0,blend_radius_m)
      movel([0.345634, -1.429666, -2.536892, -0.745831, 1.570796, 1.916430],accel_mss,speed_ms,0,blend_radius_m)
      movel([0.345544, -1.429636, -2.536915, -0.745838, 1.570796, 1.916340],accel_mss,speed_ms,0,blend_radius_m)
      movel([0.345462, -1.429597, -2.536946, -0.745847, 1.570796, 1.916259],accel_mss,speed_ms,0,blend_radius_m)
      movel([0.345395, -1.429544, -2.536987, -0.745859, 1.570796, 1.916191],accel_mss,speed_ms,0,blend_radius_m)
      movel([0.345334, -1.429474, -2.537041, -0.745874, 1.570796, 1.916130],accel_mss,speed_ms,0,blend_radius_m)
      movel([0.345282, -1.429395, -2.537102, -0.745892, 1.570796, 1.916079],accel_mss,speed_ms,0,blend_radius_m)
      movel([0.345245, -1.429310, -2.537169, -0.745911, 1.570796, 1.916041],accel_mss,speed_ms,0,blend_radius_m)
      movel([0.345220, -1.429218, -2.537240, -0.745931, 1.570796, 1.916017],accel_mss,speed_ms,0,blend_radius_m)
      movel([0.345208, -1.429119, -2.537317, -0.745953, 1.570796, 1.916004],accel_mss,speed_ms,0,blend_radius_m)
      movel([0.345210, -1.429015, -2.537398, -0.745976, 1.570796, 1.916006],accel_mss,speed_ms,0,blend_radius_m)
      movel([0.345225, -1.428907, -2.537482, -0.746000, 1.570796, 1.916021],accel_mss,speed_ms,0,blend_radius_m)
      movel([0.345253, -1.428798, -2.537566, -0.746025, 1.570796, 1.916049],accel_mss,speed_ms,0,blend_radius_m)
      movel([0.345292, -1.428696, -2.537645, -0.746047, 1.570796, 1.916088],accel_mss,speed_ms,0,blend_radius_m)
      movel([0.345346, -1.428594, -2.537724, -0.746070, 1.570796, 1.916142],accel_mss,speed_ms,0,blend_radius_m)
      movel([0.345412, -1.428496, -2.537800, -0.746092, 1.570796, 1.916208],accel_mss,speed_ms,0,blend_radius_m)
      movel([0.345491, -1.428403, -2.537872, -0.746113, 1.570796, 1.916288],accel_mss,speed_ms,0,blend_radius_m)
      movel([0.345618, -1.428273, -2.537973, -0.746142, 1.570796, 1.916414],accel_mss,speed_ms,0,blend_radius_m)
      movel([0.345757, -1.428151, -2.538068, -0.746170, 1.570796, 1.916553],accel_mss,speed_ms,0,blend_radius_m)
      movel([0.345901, -1.428039, -2.538155, -0.746195, 1.570796, 1.916697],accel_mss,speed_ms,0,blend_radius_m)
      movel([0.346001, -1.427972, -2.538207, -0.746210, 1.570796, 1.916798],accel_mss,speed_ms,0,blend_radius_m)
      movel([0.346103, -1.427914, -2.538252, -0.746223, 1.570796, 1.916899],accel_mss,speed_ms,0,blend_radius_m)
      movel([0.346209, -1.427865, -2.538290, -0.746234, 1.570796, 1.917006],accel_mss,speed_ms,0,blend_radius_m)
      movel([0.346315, -1.427825, -2.538321, -0.746243, 1.570796, 1.917111],accel_mss,speed_ms,0,blend_radius_m)
      movel([0.346415, -1.427798, -2.538342, -0.746249, 1.570796, 1.917212],accel_mss,speed_ms,0,blend_radius_m)
      movel([0.346512, -1.427782, -2.538355, -0.746253, 1.570796, 1.917308],accel_mss,speed_ms,0,blend_radius_m)
      movel([0.346606, -1.427777, -2.538358, -0.746254, 1.570796, 1.917402],accel_mss,speed_ms,0,blend_radius_m)
      movel([0.346697, -1.427782, -2.538354, -0.746253, 1.570796, 1.917493],accel_mss,speed_ms,0,blend_radius_m)
      speed_ms = 0.003
      movel([0.346697, -1.415265, -2.532641, -0.764483, 1.570796, 1.917493],accel_mss,speed_ms,0,blend_radius_m)
      speed_ms = 0.01
      movel([0.346697, -1.391181, -2.520822, -0.800386, 1.570796, 1.917493],accel_mss,speed_ms,0,blend_radius_m)
      movel([0.314052, -1.382109, -2.527415, -0.802865, 1.570796, 1.884848],accel_mss,speed_ms,0,blend_radius_m)
      movel([0.314052, -1.406365, -2.539347, -0.766677, 1.570796, 1.884848],accel_mss,speed_ms,0,blend_radius_m)
      speed_ms = 0.003
      movel([0.314052, -1.415796, -2.543687, -0.752906, 1.570796, 1.884848],accel_mss,speed_ms,0,blend_radius_m)
      speed_ms = 0.007
      movel([0.313677, -1.416288, -2.543314, -0.752788, 1.570796, 1.884473],accel_mss,speed_ms,0,blend_radius_m)
      movel([0.313291, -1.416774, -2.542945, -0.752670, 1.570796, 1.884087],accel_mss,speed_ms,0,blend_radius_m)
      movel([0.312894, -1.417254, -2.542580, -0.752555, 1.570796, 1.883690],accel_mss,speed_ms,0,blend_radius_m)
      movel([0.312488, -1.417728, -2.542219, -0.752441, 1.570796, 1.883284],accel_mss,speed_ms,0,blend_radius_m)
      movel([0.312070, -1.418197, -2.541862, -0.752329, 1.570796, 1.882867],accel_mss,speed_ms,0,blend_radius_m)
      movel([0.311650, -1.418652, -2.541516, -0.752221, 1.570796, 1.882446],accel_mss,speed_ms,0,blend_radius_m)
      movel([0.311220, -1.419100, -2.541174, -0.752115, 1.570796, 1.882017],accel_mss,speed_ms,0,blend_radius_m)
      movel([0.310783, -1.419541, -2.540838, -0.752010, 1.570796, 1.881579],accel_mss,speed_ms,0,blend_radius_m)
      movel([0.310335, -1.419974, -2.540507, -0.751908, 1.570796, 1.881131],accel_mss,speed_ms,0,blend_radius_m)
      movel([0.309878, -1.420401, -2.540180, -0.751807, 1.570796, 1.880674],accel_mss,speed_ms,0,blend_radius_m)
      movel([0.309414, -1.420819, -2.539861, -0.751709, 1.570796, 1.880210],accel_mss,speed_ms,0,blend_radius_m)
      movel([0.308942, -1.421228, -2.539547, -0.751613, 1.570796, 1.879738],accel_mss,speed_ms,0,blend_radius_m)
      movel([0.308461, -1.421630, -2.539240, -0.751519, 1.570796, 1.879258],accel_mss,speed_ms,0,blend_radius_m)
      movel([0.307976, -1.422022, -2.538939, -0.751428, 1.570796, 1.878772],accel_mss,speed_ms,0,blend_radius_m)
      movel([0.307480, -1.422406, -2.538644, -0.751339, 1.570796, 1.878276],accel_mss,speed_ms,0,blend_radius_m)
      movel([0.307008, -1.422760, -2.538373, -0.751257, 1.570796, 1.877805],accel_mss,speed_ms,0,blend_radius_m)
      movel([0.306532, -1.423107, -2.538106, -0.751176, 1.570796, 1.877329],accel_mss,speed_ms,0,blend_radius_m)
      movel([0.306049, -1.423445, -2.537846, -0.751098, 1.570796, 1.876845],accel_mss,speed_ms,0,blend_radius_m)
      movel([0.305564, -1.423775, -2.537592, -0.751022, 1.570796, 1.876360],accel_mss,speed_ms,0,blend_radius_m)
      movel([0.305072, -1.424099, -2.537343, -0.750948, 1.570796, 1.875869],accel_mss,speed_ms,0,blend_radius_m)
      movel([0.304596, -1.424399, -2.537111, -0.750879, 1.570796, 1.875392],accel_mss,speed_ms,0,blend_radius_m)
      movel([0.304118, -1.424689, -2.536888, -0.750813, 1.570796, 1.874915],accel_mss,speed_ms,0,blend_radius_m)
      movel([0.303635, -1.424971, -2.536670, -0.750748, 1.570796, 1.874431],accel_mss,speed_ms,0,blend_radius_m)
      movel([0.303149, -1.425243, -2.536460, -0.750686, 1.570796, 1.873945],accel_mss,speed_ms,0,blend_radius_m)
      movel([0.302659, -1.425505, -2.536258, -0.750626, 1.570796, 1.873456],accel_mss,speed_ms,0,blend_radius_m)
      movel([0.302165, -1.425758, -2.536062, -0.750569, 1.570796, 1.872961],accel_mss,speed_ms,0,blend_radius_m)
      movel([0.301669, -1.426000, -2.535875, -0.750514, 1.570796, 1.872465],accel_mss,speed_ms,0,blend_radius_m)
      movel([0.301171, -1.426233, -2.535695, -0.750461, 1.570796, 1.871967],accel_mss,speed_ms,0,blend_radius_m)
      movel([0.300669, -1.426455, -2.535523, -0.750411, 1.570796, 1.871465],accel_mss,speed_ms,0,blend_radius_m)
      movel([0.300169, -1.426666, -2.535360, -0.750363, 1.570796, 1.870966],accel_mss,speed_ms,0,blend_radius_m)
      movel([0.299643, -1.426876, -2.535197, -0.750316, 1.570796, 1.870440],accel_mss,speed_ms,0,blend_radius_m)
      movel([0.299116, -1.427077, -2.535042, -0.750270, 1.570796, 1.869913],accel_mss,speed_ms,0,blend_radius_m)
      movel([0.298589, -1.427268, -2.534894, -0.750227, 1.570796, 1.869385],accel_mss,speed_ms,0,blend_radius_m)
      movel([0.298060, -1.427448, -2.534754, -0.750187, 1.570796, 1.868856],accel_mss,speed_ms,0,blend_radius_m)
      movel([0.297533, -1.427619, -2.534622, -0.750149, 1.570796, 1.868329],accel_mss,speed_ms,0,blend_radius_m)
      movel([0.297159, -1.427731, -2.534535, -0.750123, 1.570796, 1.867955],accel_mss,speed_ms,0,blend_radius_m)
      movel([0.296785, -1.427831, -2.534457, -0.750101, 1.570796, 1.867581],accel_mss,speed_ms,0,blend_radius_m)
      movel([0.296415, -1.427919, -2.534389, -0.750081, 1.570796, 1.867211],accel_mss,speed_ms,0,blend_radius_m)
      movel([0.296044, -1.427996, -2.534329, -0.750064, 1.570796, 1.866840],accel_mss,speed_ms,0,blend_radius_m)
      movel([0.295677, -1.428062, -2.534278, -0.750049, 1.570796, 1.866474],accel_mss,speed_ms,0,blend_radius_m)
      movel([0.295078, -1.428152, -2.534208, -0.750029, 1.570796, 1.865874],accel_mss,speed_ms,0,blend_radius_m)
      movel([0.294481, -1.428234, -2.534145, -0.750011, 1.570796, 1.865278],accel_mss,speed_ms,0,blend_radius_m)
      movel([0.293889, -1.428303, -2.534090, -0.749995, 1.570796, 1.864685],accel_mss,speed_ms,0,blend_radius_m)
      movel([0.293298, -1.428361, -2.534046, -0.749982, 1.570796, 1.864095],accel_mss,speed_ms,0,blend_radius_m)
      movel([0.292712, -1.428410, -2.534007, -0.749971, 1.570796, 1.863509],accel_mss,speed_ms,0,blend_radius_m)
      movel([0.292131, -1.428447, -2.533979, -0.749963, 1.570796, 1.862927],accel_mss,speed_ms,0,blend_radius_m)
      movel([0.291553, -1.428472, -2.533960, -0.749958, 1.570796, 1.862349],accel_mss,speed_ms,0,blend_radius_m)
      movel([0.290978, -1.428488, -2.533947, -0.749954, 1.570796, 1.861774],accel_mss,speed_ms,0,blend_radius_m)
      movel([0.290633, -1.428488, -2.533947, -0.749954, 1.570796, 1.861429],accel_mss,speed_ms,0,blend_radius_m)
      movel([0.290291, -1.428475, -2.533957, -0.749957, 1.570796, 1.861088],accel_mss,speed_ms,0,blend_radius_m)
      movel([0.289956, -1.428452, -2.533975, -0.749962, 1.570796, 1.860752],accel_mss,speed_ms,0,blend_radius_m)
      movel([0.289629, -1.428415, -2.534003, -0.749970, 1.570796, 1.860425],accel_mss,speed_ms,0,blend_radius_m)
      movel([0.289306, -1.428366, -2.534041, -0.749981, 1.570796, 1.860102],accel_mss,speed_ms,0,blend_radius_m)
      movel([0.288849, -1.428282, -2.534107, -0.750000, 1.570796, 1.859645],accel_mss,speed_ms,0,blend_radius_m)
      movel([0.288400, -1.428186, -2.534182, -0.750021, 1.570796, 1.859196],accel_mss,speed_ms,0,blend_radius_m)
      movel([0.287956, -1.428080, -2.534264, -0.750045, 1.570796, 1.858752],accel_mss,speed_ms,0,blend_radius_m)
      movel([0.287522, -1.427963, -2.534355, -0.750071, 1.570796, 1.858319],accel_mss,speed_ms,0,blend_radius_m)
      movel([0.287095, -1.427833, -2.534455, -0.750100, 1.570796, 1.857891],accel_mss,speed_ms,0,blend_radius_m)
      movel([0.286701, -1.427703, -2.534557, -0.750130, 1.570796, 1.857497],accel_mss,speed_ms,0,blend_radius_m)
      movel([0.286315, -1.427557, -2.534670, -0.750162, 1.570796, 1.857112],accel_mss,speed_ms,0,blend_radius_m)
      movel([0.285940, -1.427400, -2.534791, -0.750198, 1.570796, 1.856736],accel_mss,speed_ms,0,blend_radius_m)
      movel([0.285575, -1.427233, -2.534921, -0.750235, 1.570796, 1.856371],accel_mss,speed_ms,0,blend_radius_m)
      movel([0.285220, -1.427052, -2.535061, -0.750276, 1.570796, 1.856016],accel_mss,speed_ms,0,blend_radius_m)
      movel([0.284876, -1.426858, -2.535211, -0.750320, 1.570796, 1.855672],accel_mss,speed_ms,0,blend_radius_m)
      movel([0.284542, -1.426653, -2.535370, -0.750366, 1.570796, 1.855338],accel_mss,speed_ms,0,blend_radius_m)
      movel([0.284217, -1.426437, -2.535537, -0.750415, 1.570796, 1.855014],accel_mss,speed_ms,0,blend_radius_m)
      movel([0.283905, -1.426210, -2.535713, -0.750466, 1.570796, 1.854702],accel_mss,speed_ms,0,blend_radius_m)
      movel([0.283606, -1.425971, -2.535898, -0.750520, 1.570796, 1.854402],accel_mss,speed_ms,0,blend_radius_m)
      movel([0.283296, -1.425707, -2.536102, -0.750580, 1.570796, 1.854092],accel_mss,speed_ms,0,blend_radius_m)
      movel([0.282998, -1.425433, -2.536313, -0.750643, 1.570796, 1.853794],accel_mss,speed_ms,0,blend_radius_m)
      movel([0.282710, -1.425149, -2.536533, -0.750707, 1.570796, 1.853506],accel_mss,speed_ms,0,blend_radius_m)
      movel([0.282433, -1.424855, -2.536760, -0.750775, 1.570796, 1.853230],accel_mss,speed_ms,0,blend_radius_m)
      movel([0.282168, -1.424553, -2.536992, -0.750843, 1.570796, 1.852964],accel_mss,speed_ms,0,blend_radius_m)
      movel([0.281908, -1.424231, -2.537240, -0.750917, 1.570796, 1.852705],accel_mss,speed_ms,0,blend_radius_m)
      movel([0.281660, -1.423902, -2.537494, -0.750993, 1.570796, 1.852456],accel_mss,speed_ms,0,blend_radius_m)
      movel([0.281424, -1.423561, -2.537757, -0.751072, 1.570796, 1.852220],accel_mss,speed_ms,0,blend_radius_m)
      movel([0.281204, -1.423210, -2.538027, -0.751153, 1.570796, 1.852000],accel_mss,speed_ms,0,blend_radius_m)
      movel([0.280995, -1.422851, -2.538302, -0.751235, 1.570796, 1.851791],accel_mss,speed_ms,0,blend_radius_m)
      movel([0.280805, -1.422489, -2.538581, -0.751319, 1.570796, 1.851601],accel_mss,speed_ms,0,blend_radius_m)
      movel([0.280628, -1.422119, -2.538865, -0.751405, 1.570796, 1.851424],accel_mss,speed_ms,0,blend_radius_m)
      movel([0.280467, -1.421739, -2.539156, -0.751494, 1.570796, 1.851263],accel_mss,speed_ms,0,blend_radius_m)
      movel([0.280320, -1.421349, -2.539455, -0.751585, 1.570796, 1.851116],accel_mss,speed_ms,0,blend_radius_m)
      movel([0.280187, -1.420951, -2.539760, -0.751678, 1.570796, 1.850983],accel_mss,speed_ms,0,blend_radius_m)
      movel([0.280067, -1.420537, -2.540076, -0.751775, 1.570796, 1.850863],accel_mss,speed_ms,0,blend_radius_m)
      movel([0.279961, -1.420114, -2.540400, -0.751875, 1.570796, 1.850757],accel_mss,speed_ms,0,blend_radius_m)
      movel([0.279870, -1.419685, -2.540728, -0.751976, 1.570796, 1.850667],accel_mss,speed_ms,0,blend_radius_m)
      movel([0.279795, -1.419247, -2.541062, -0.752080, 1.570796, 1.850592],accel_mss,speed_ms,0,blend_radius_m)
      movel([0.279735, -1.418804, -2.541400, -0.752185, 1.570796, 1.850532],accel_mss,speed_ms,0,blend_radius_m)
      movel([0.279686, -1.418324, -2.541766, -0.752299, 1.570796, 1.850483],accel_mss,speed_ms,0,blend_radius_m)
      movel([0.279652, -1.417840, -2.542134, -0.752415, 1.570796, 1.850448],accel_mss,speed_ms,0,blend_radius_m)
      movel([0.279628, -1.417351, -2.542506, -0.752532, 1.570796, 1.850424],accel_mss,speed_ms,0,blend_radius_m)
      movel([0.279622, -1.416853, -2.542884, -0.752651, 1.570796, 1.850419],accel_mss,speed_ms,0,blend_radius_m)
      movel([0.279626, -1.416354, -2.543263, -0.752771, 1.570796, 1.850422],accel_mss,speed_ms,0,blend_radius_m)
      movel([0.279638, -1.416064, -2.543483, -0.752841, 1.570796, 1.850434],accel_mss,speed_ms,0,blend_radius_m)
      movel([0.279658, -1.415769, -2.543707, -0.752913, 1.570796, 1.850454],accel_mss,speed_ms,0,blend_radius_m)
      movel([0.279687, -1.415475, -2.543930, -0.752984, 1.570796, 1.850483],accel_mss,speed_ms,0,blend_radius_m)
      movel([0.279726, -1.415198, -2.544139, -0.753051, 1.570796, 1.850522],accel_mss,speed_ms,0,blend_radius_m)
      movel([0.279771, -1.414923, -2.544348, -0.753118, 1.570796, 1.850568],accel_mss,speed_ms,0,blend_radius_m)
      movel([0.279832, -1.414642, -2.544561, -0.753187, 1.570796, 1.850628],accel_mss,speed_ms,0,blend_radius_m)
      movel([0.279917, -1.414283, -2.544832, -0.753274, 1.570796, 1.850713],accel_mss,speed_ms,0,blend_radius_m)
      movel([0.280011, -1.413921, -2.545105, -0.753363, 1.570796, 1.850808],accel_mss,speed_ms,0,blend_radius_m)
      movel([0.280115, -1.413560, -2.545377, -0.753451, 1.570796, 1.850911],accel_mss,speed_ms,0,blend_radius_m)
      movel([0.280391, -1.412635, -2.546075, -0.753679, 1.570796, 1.851188],accel_mss,speed_ms,0,blend_radius_m)
      movel([0.280678, -1.411708, -2.546772, -0.753908, 1.570796, 1.851474],accel_mss,speed_ms,0,blend_radius_m)
      movel([0.280987, -1.410738, -2.547501, -0.754150, 1.570796, 1.851783],accel_mss,speed_ms,0,blend_radius_m)
      movel([0.281302, -1.409763, -2.548232, -0.754394, 1.570796, 1.852098],accel_mss,speed_ms,0,blend_radius_m)
      movel([0.281425, -1.409404, -2.548501, -0.754484, 1.570796, 1.852222],accel_mss,speed_ms,0,blend_radius_m)
      movel([0.281559, -1.409042, -2.548772, -0.754575, 1.570796, 1.852355],accel_mss,speed_ms,0,blend_radius_m)
      movel([0.281701, -1.408680, -2.549042, -0.754667, 1.570796, 1.852497],accel_mss,speed_ms,0,blend_radius_m)
      movel([0.281827, -1.408385, -2.549263, -0.754741, 1.570796, 1.852623],accel_mss,speed_ms,0,blend_radius_m)
      movel([0.281964, -1.408090, -2.549483, -0.754816, 1.570796, 1.852760],accel_mss,speed_ms,0,blend_radius_m)
      movel([0.282113, -1.407794, -2.549704, -0.754891, 1.570796, 1.852909],accel_mss,speed_ms,0,blend_radius_m)
      movel([0.282407, -1.407251, -2.550109, -0.755029, 1.570796, 1.853203],accel_mss,speed_ms,0,blend_radius_m)
      movel([0.282716, -1.406709, -2.550513, -0.755167, 1.570796, 1.853512],accel_mss,speed_ms,0,blend_radius_m)
      movel([0.283060, -1.406138, -2.550938, -0.755314, 1.570796, 1.853856],accel_mss,speed_ms,0,blend_radius_m)
      movel([0.283416, -1.405569, -2.551360, -0.755460, 1.570796, 1.854213],accel_mss,speed_ms,0,blend_radius_m)
      movel([0.283790, -1.405004, -2.551780, -0.755605, 1.570796, 1.854586],accel_mss,speed_ms,0,blend_radius_m)
      movel([0.284177, -1.404442, -2.552197, -0.755751, 1.570796, 1.854973],accel_mss,speed_ms,0,blend_radius_m)
      movel([0.284577, -1.403881, -2.552612, -0.755896, 1.570796, 1.855373],accel_mss,speed_ms,0,blend_radius_m)
      movel([0.284991, -1.403328, -2.553021, -0.756040, 1.570796, 1.855787],accel_mss,speed_ms,0,blend_radius_m)
      movel([0.285421, -1.402776, -2.553429, -0.756184, 1.570796, 1.856217],accel_mss,speed_ms,0,blend_radius_m)
      movel([0.285863, -1.402229, -2.553833, -0.756327, 1.570796, 1.856659],accel_mss,speed_ms,0,blend_radius_m)
      movel([0.286317, -1.401689, -2.554231, -0.756469, 1.570796, 1.857113],accel_mss,speed_ms,0,blend_radius_m)
      movel([0.286768, -1.401172, -2.554612, -0.756605, 1.570796, 1.857565],accel_mss,speed_ms,0,blend_radius_m)
      movel([0.287233, -1.400663, -2.554986, -0.756739, 1.570796, 1.858030],accel_mss,speed_ms,0,blend_radius_m)
      movel([0.287711, -1.400160, -2.555357, -0.756873, 1.570796, 1.858507],accel_mss,speed_ms,0,blend_radius_m)
      movel([0.288202, -1.399665, -2.555720, -0.757004, 1.570796, 1.858998],accel_mss,speed_ms,0,blend_radius_m)
      movel([0.288701, -1.399180, -2.556076, -0.757133, 1.570796, 1.859498],accel_mss,speed_ms,0,blend_radius_m)
      movel([0.289215, -1.398701, -2.556427, -0.757261, 1.570796, 1.860011],accel_mss,speed_ms,0,blend_radius_m)
      movel([0.289741, -1.398229, -2.556773, -0.757387, 1.570796, 1.860537],accel_mss,speed_ms,0,blend_radius_m)
      movel([0.290274, -1.397769, -2.557109, -0.757511, 1.570796, 1.861071],accel_mss,speed_ms,0,blend_radius_m)
      movel([0.290819, -1.397318, -2.557439, -0.757632, 1.570796, 1.861615],accel_mss,speed_ms,0,blend_radius_m)
      movel([0.291362, -1.396889, -2.557752, -0.757748, 1.570796, 1.862158],accel_mss,speed_ms,0,blend_radius_m)
      movel([0.291912, -1.396467, -2.558060, -0.757862, 1.570796, 1.862708],accel_mss,speed_ms,0,blend_radius_m)
      movel([0.292474, -1.396059, -2.558358, -0.757972, 1.570796, 1.863270],accel_mss,speed_ms,0,blend_radius_m)
      movel([0.293042, -1.395660, -2.558648, -0.758080, 1.570796, 1.863838],accel_mss,speed_ms,0,blend_radius_m)
      movel([0.293615, -1.395276, -2.558928, -0.758185, 1.570796, 1.864411],accel_mss,speed_ms,0,blend_radius_m)
      movel([0.294199, -1.394901, -2.559200, -0.758287, 1.570796, 1.864995],accel_mss,speed_ms,0,blend_radius_m)
      movel([0.294788, -1.394541, -2.559462, -0.758385, 1.570796, 1.865584],accel_mss,speed_ms,0,blend_radius_m)
      movel([0.295381, -1.394196, -2.559713, -0.758480, 1.570796, 1.866177],accel_mss,speed_ms,0,blend_radius_m)
      movel([0.295981, -1.393860, -2.559957, -0.758572, 1.570796, 1.866777],accel_mss,speed_ms,0,blend_radius_m)
      movel([0.296585, -1.393541, -2.560188, -0.758660, 1.570796, 1.867381],accel_mss,speed_ms,0,blend_radius_m)
      movel([0.297191, -1.393235, -2.560410, -0.758744, 1.570796, 1.867988],accel_mss,speed_ms,0,blend_radius_m)
      movel([0.297803, -1.392943, -2.560622, -0.758824, 1.570796, 1.868599],accel_mss,speed_ms,0,blend_radius_m)
      movel([0.298417, -1.392666, -2.560822, -0.758901, 1.570796, 1.869213],accel_mss,speed_ms,0,blend_radius_m)
      movel([0.299033, -1.392405, -2.561012, -0.758973, 1.570796, 1.869829],accel_mss,speed_ms,0,blend_radius_m)
      movel([0.299650, -1.392160, -2.561188, -0.759041, 1.570796, 1.870446],accel_mss,speed_ms,0,blend_radius_m)
      movel([0.300268, -1.391928, -2.561356, -0.759105, 1.570796, 1.871064],accel_mss,speed_ms,0,blend_radius_m)
      movel([0.300887, -1.391714, -2.561511, -0.759164, 1.570796, 1.871684],accel_mss,speed_ms,0,blend_radius_m)
      movel([0.301504, -1.391515, -2.561655, -0.759219, 1.570796, 1.872301],accel_mss,speed_ms,0,blend_radius_m)
      movel([0.302008, -1.391368, -2.561761, -0.759260, 1.570796, 1.872804],accel_mss,speed_ms,0,blend_radius_m)
      movel([0.302511, -1.391237, -2.561856, -0.759297, 1.570796, 1.873307],accel_mss,speed_ms,0,blend_radius_m)
      movel([0.303009, -1.391121, -2.561939, -0.759329, 1.570796, 1.873805],accel_mss,speed_ms,0,blend_radius_m)
      movel([0.303506, -1.391023, -2.562010, -0.759356, 1.570796, 1.874302],accel_mss,speed_ms,0,blend_radius_m)
      movel([0.304074, -1.390924, -2.562081, -0.759384, 1.570796, 1.874870],accel_mss,speed_ms,0,blend_radius_m)
      movel([0.304640, -1.390839, -2.562142, -0.759407, 1.570796, 1.875436],accel_mss,speed_ms,0,blend_radius_m)
      movel([0.305199, -1.390768, -2.562194, -0.759427, 1.570796, 1.875995],accel_mss,speed_ms,0,blend_radius_m)
      movel([0.305757, -1.390708, -2.562237, -0.759444, 1.570796, 1.876553],accel_mss,speed_ms,0,blend_radius_m)
      movel([0.306310, -1.390661, -2.562271, -0.759457, 1.570796, 1.877106],accel_mss,speed_ms,0,blend_radius_m)
      movel([0.306859, -1.390626, -2.562296, -0.759467, 1.570796, 1.877656],accel_mss,speed_ms,0,blend_radius_m)
      movel([0.307404, -1.390604, -2.562312, -0.759473, 1.570796, 1.878200],accel_mss,speed_ms,0,blend_radius_m)
      movel([0.307942, -1.390597, -2.562317, -0.759475, 1.570796, 1.878738],accel_mss,speed_ms,0,blend_radius_m)
      movel([0.308401, -1.390603, -2.562313, -0.759473, 1.570796, 1.879198],accel_mss,speed_ms,0,blend_radius_m)
      movel([0.308855, -1.390628, -2.562295, -0.759466, 1.570796, 1.879651],accel_mss,speed_ms,0,blend_radius_m)
      movel([0.309299, -1.390668, -2.562266, -0.759455, 1.570796, 1.880095],accel_mss,speed_ms,0,blend_radius_m)
      movel([0.309734, -1.390725, -2.562225, -0.759439, 1.570796, 1.880531],accel_mss,speed_ms,0,blend_radius_m)
      movel([0.310264, -1.390816, -2.562159, -0.759414, 1.570796, 1.881060],accel_mss,speed_ms,0,blend_radius_m)
      movel([0.310782, -1.390924, -2.562081, -0.759384, 1.570796, 1.881579],accel_mss,speed_ms,0,blend_radius_m)
      movel([0.311288, -1.391050, -2.561990, -0.759349, 1.570796, 1.882084],accel_mss,speed_ms,0,blend_radius_m)
      movel([0.311782, -1.391195, -2.561885, -0.759308, 1.570796, 1.882578],accel_mss,speed_ms,0,blend_radius_m)
      movel([0.312265, -1.391354, -2.561771, -0.759264, 1.570796, 1.883061],accel_mss,speed_ms,0,blend_radius_m)
      movel([0.312730, -1.391535, -2.561640, -0.759214, 1.570796, 1.883527],accel_mss,speed_ms,0,blend_radius_m)
      movel([0.313189, -1.391729, -2.561500, -0.759160, 1.570796, 1.883985],accel_mss,speed_ms,0,blend_radius_m)
      movel([0.313630, -1.391942, -2.561346, -0.759101, 1.570796, 1.884426],accel_mss,speed_ms,0,blend_radius_m)
      movel([0.314058, -1.392169, -2.561182, -0.759038, 1.570796, 1.884854],accel_mss,speed_ms,0,blend_radius_m)
      movel([0.314471, -1.392415, -2.561004, -0.758970, 1.570796, 1.885267],accel_mss,speed_ms,0,blend_radius_m)
      movel([0.314869, -1.392675, -2.560816, -0.758898, 1.570796, 1.885665],accel_mss,speed_ms,0,blend_radius_m)
      movel([0.315252, -1.392952, -2.560615, -0.758822, 1.570796, 1.886049],accel_mss,speed_ms,0,blend_radius_m)
      movel([0.315618, -1.393246, -2.560403, -0.758741, 1.570796, 1.886415],accel_mss,speed_ms,0,blend_radius_m)
      movel([0.315972, -1.393553, -2.560180, -0.758656, 1.570796, 1.886768],accel_mss,speed_ms,0,blend_radius_m)
      movel([0.316307, -1.393875, -2.559946, -0.758568, 1.570796, 1.887103],accel_mss,speed_ms,0,blend_radius_m)
      movel([0.316625, -1.394212, -2.559702, -0.758476, 1.570796, 1.887421],accel_mss,speed_ms,0,blend_radius_m)
      movel([0.316927, -1.394562, -2.559447, -0.758380, 1.570796, 1.887723],accel_mss,speed_ms,0,blend_radius_m)
      movel([0.317209, -1.394927, -2.559182, -0.758280, 1.570796, 1.888006],accel_mss,speed_ms,0,blend_radius_m)
      movel([0.317478, -1.395307, -2.558906, -0.758177, 1.570796, 1.888274],accel_mss,speed_ms,0,blend_radius_m)
      movel([0.317727, -1.395700, -2.558619, -0.758070, 1.570796, 1.888523],accel_mss,speed_ms,0,blend_radius_m)
      movel([0.317959, -1.396104, -2.558325, -0.757960, 1.570796, 1.888756],accel_mss,speed_ms,0,blend_radius_m)
      movel([0.318170, -1.396522, -2.558020, -0.757847, 1.570796, 1.888966],accel_mss,speed_ms,0,blend_radius_m)
      movel([0.318366, -1.396949, -2.557708, -0.757731, 1.570796, 1.889162],accel_mss,speed_ms,0,blend_radius_m)
      movel([0.318541, -1.397389, -2.557387, -0.757613, 1.570796, 1.889338],accel_mss,speed_ms,0,blend_radius_m)
      movel([0.318684, -1.397780, -2.557101, -0.757508, 1.570796, 1.889480],accel_mss,speed_ms,0,blend_radius_m)
      movel([0.318813, -1.398180, -2.556808, -0.757400, 1.570796, 1.889610],accel_mss,speed_ms,0,blend_radius_m)
      movel([0.318930, -1.398586, -2.556511, -0.757292, 1.570796, 1.889726],accel_mss,speed_ms,0,blend_radius_m)
      movel([0.319035, -1.398997, -2.556210, -0.757182, 1.570796, 1.889832],accel_mss,speed_ms,0,blend_radius_m)
      movel([0.319122, -1.399383, -2.555927, -0.757079, 1.570796, 1.889918],accel_mss,speed_ms,0,blend_radius_m)
      movel([0.319192, -1.399776, -2.555638, -0.756974, 1.570796, 1.889989],accel_mss,speed_ms,0,blend_radius_m)
      movel([0.319252, -1.400175, -2.555345, -0.756868, 1.570796, 1.890048],accel_mss,speed_ms,0,blend_radius_m)
      movel([0.319295, -1.400581, -2.555047, -0.756761, 1.570796, 1.890091],accel_mss,speed_ms,0,blend_radius_m)
      movel([0.319326, -1.401001, -2.554738, -0.756650, 1.570796, 1.890123],accel_mss,speed_ms,0,blend_radius_m)
      movel([0.319344, -1.401428, -2.554424, -0.756537, 1.570796, 1.890140],accel_mss,speed_ms,0,blend_radius_m)
      movel([0.319347, -1.401858, -2.554107, -0.756424, 1.570796, 1.890143],accel_mss,speed_ms,0,blend_radius_m)
      movel([0.319338, -1.402295, -2.553784, -0.756310, 1.570796, 1.890134],accel_mss,speed_ms,0,blend_radius_m)
      movel([0.319303, -1.402955, -2.553297, -0.756137, 1.570796, 1.890099],accel_mss,speed_ms,0,blend_radius_m)
      movel([0.319250, -1.403620, -2.552805, -0.755964, 1.570796, 1.890046],accel_mss,speed_ms,0,blend_radius_m)
      movel([0.319177, -1.404290, -2.552309, -0.755790, 1.570796, 1.889973],accel_mss,speed_ms,0,blend_radius_m)
      movel([0.319122, -1.404672, -2.552026, -0.755691, 1.570796, 1.889918],accel_mss,speed_ms,0,blend_radius_m)
      movel([0.319055, -1.405054, -2.551743, -0.755592, 1.570796, 1.889852],accel_mss,speed_ms,0,blend_radius_m)
      movel([0.318973, -1.405442, -2.551455, -0.755492, 1.570796, 1.889770],accel_mss,speed_ms,0,blend_radius_m)
      movel([0.318880, -1.405830, -2.551166, -0.755393, 1.570796, 1.889676],accel_mss,speed_ms,0,blend_radius_m)
